KUKA KRL program: EPS_2_251674_SAN03_A_20251204014858.src

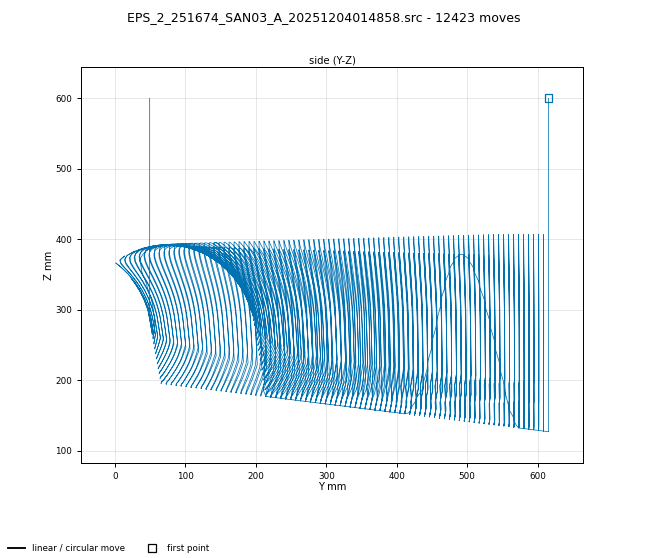
[picture p0: tool path of EPS_2_251674_SAN03_A_20251204014858.src, 12423 of 12425 moves have a stored position in this frame; points joined in program order, loops and branches not executed]
&ACCESS RVP
&REL 4
&COMMENT QRS 19112012
&PARAM EDITMASK = *
DEF PART()
EXT BAS (BAS_COMMAND :IN,REAL :IN )
INT I
BAS (#INITMOV,0 )

;KUKA QRS Post kuka4.cps  Date:22-06-2017 !

File_ID=2940

QRS_PRE_INIT()

;Init var - Until changes are made in qrs_pre_init
Outlet_Square_prg=0
Inlet_1_Square_prg=0
Inlet_2_Square_prg=0
Inlet_3_Square_prg=0
Inlet_4_Square_prg=0
Inlet_5_Square_prg=0

Outlet_1={X 0.000, Y 546.330, Z 306.500, B 0.000, E1 0.000 }
Inlet_1={X 0.000, Y 548.460, Z 276.500, B 0.000, E1 134.000 }
Outlet_1_type=201
Inlet_1_type=201
;QRS#1=Sidecore dimensions
;QRS#2=200-8" PVC SDR 35
;QRS#3=200-8" PVC SDR 35
;QRS#4=
;QRS#5=
;QRS#6=
;QRS#7=
;QRS#8=
;QRS#9=12-08 PSX
;QRS#10=12-08 PSX
;QRS#11=
;QRS#12=
;QRS#13=
;QRS#14=
;QRS#15=
;QRS#16=1220x127x686 2,25'
;QRS#17=EPS Height
;QRS#18=407
;QRS#19=*
;QRS#20= UPDATED VERSION 22-06-2017
;QRS#21=*
Outlet_Square=0100
Inlet_1_Square=0100
Inlet_2_Square=0
Inlet_3_Square=0
Inlet_4_Square=0
Inlet_5_Square=0
Mill_Square=1
Outlet_Square_Prg=204
Inlet_1_Square_prg=204

QRS_INIT()

$ADVANCE=5

; T1
PTP {E1 173.652,E2 173.652}
PTP {X 0,Y 615.437,A -85,B 0,C 180,E1 173.652,E2 173.652,E3 0,E4 0,E5 0,E6 0}
QRS_SPEED_INIT()
LIN {X 0,Y 615.437,Z 600,A -85,B 0,C 180,E1 173.652,E2 173.652,E3 0,E4 0,E5 0,E6 0} C_VEL
LIN {X 0,Y 615.437,Z 136.877,A -85,B 0,C 180,E1 173.652,E2 173.652} C_VEL
LIN {X 0,Y 615.437,Z 128.699,A -85,B 0,C 180,E1 173.652,E2 173.652} C_VEL
LIN {X 0,Y 615.423,Z 126.699,A -85,B 0,C 180,E1 173.466,E2 173.466} C_VEL
LIN {X 0,Y 615.421,Z 126.699,A -85,B 0,C 180,E1 171.463,E2 171.463} C_VEL
LIN {X 0,Y 615.417,Z 126.699,A -85,B 0,C 180,E1 169.141,E2 169.141} C_VEL
LIN {X 0,Y 615.44,Z 126.7,A -85,B 0,C 180,E1 166.798,E2 166.798} C_VEL
LIN {X 0,Y 615.461,Z 126.698,A -85,B 0,C 180,E1 164.094,E2 164.094} C_VEL
LIN {X 0,Y 615.415,Z 126.699,A -85,B 0,C 180,E1 161.352,E2 161.352} C_VEL
LIN {X 0,Y 615.494,Z 126.7,A -85,B 0,C 180,E1 158.569,E2 158.569} C_VEL
LIN {X 0,Y 615.418,Z 126.699,A -85,B 0,C 180,E1 155.725,E2 155.725} C_VEL
LIN {X 0,Y 615.429,Z 126.888,A -85,B 0,C 180,E1 155.186,E2 155.186} C_VEL
LIN {X 0,Y 615.495,Z 142.358,A -85,B 0,C 180,E1 152.64,E2 152.64} C_VEL
LIN {X 0,Y 615.484,Z 160.778,A -85,B 0,C 180,E1 149.651,E2 149.651} C_VEL
LIN {X 0,Y 615.49,Z 165.938,A -85,B 0,C 180,E1 148.82,E2 148.82} C_VEL
LIN {X 0,Y 615.49,Z 272.899,A -85,B 0,C 180,E1 147.543,E2 147.543} C_VEL
LIN {X 0,Y 615.48,Z 286.149,A -85,B 0,C 180,E1 147.251,E2 147.251} C_VEL
LIN {X 0,Y 615.485,Z 298.089,A -85,B 0,C 180,E1 146.862,E2 146.862} C_VEL
LIN {X 0,Y 615.469,Z 309.932,A -85,B 0,C 180,E1 146.343,E2 146.343} C_VEL
LIN {X 0,Y 615.468,Z 320.918,A -85,B 0,C 180,E1 145.722,E2 145.722} C_VEL
LIN {X 0,Y 615.498,Z 331.305,A -85,B 0,C 180,E1 144.987,E2 144.987} C_VEL
LIN {X 0,Y 615.497,Z 340.782,A -85,B 0,C 180,E1 144.164,E2 144.164} C_VEL
LIN {X 0,Y 615.498,Z 348.744,A -85,B 0,C 180,E1 143.319,E2 143.319} C_VEL
LIN {X 0,Y 615.496,Z 356.025,A -85,B 0,C 180,E1 142.373,E2 142.373} C_VEL
LIN {X 0,Y 615.493,Z 362.602,A -85,B 0,C 180,E1 141.306,E2 141.306} C_VEL
LIN {X 0,Y 615.493,Z 367.683,A -85,B 0,C 180,E1 140.251,E2 140.251} C_VEL
LIN {X 0,Y 615.494,Z 370.866,A -85,B 0,C 180,E1 139.394,E2 139.394} C_VEL
LIN {X 0,Y 615.496,Z 373.343,A -85,B 0,C 180,E1 138.527,E2 138.527} C_VEL
LIN {X 0,Y 615.499,Z 375.057,A -85,B 0,C 180,E1 137.648,E2 137.648} C_VEL
LIN {X 0,Y 615.498,Z 376.069,A -85,B 0,C 180,E1 136.757,E2 136.757} C_VEL
LIN {X 0,Y 615.496,Z 376.37,A -85,B 0,C 180,E1 135.852,E2 135.852} C_VEL
LIN {X 0,Y 615.496,Z 375.91,A -85,B 0,C 180,E1 134.933,E2 134.933} C_VEL
LIN {X 0,Y 615.493,Z 374.62,A -85,B 0,C 180,E1 133.998,E2 133.998} C_VEL
LIN {X 0,Y 615.494,Z 372.461,A -85,B 0,C 180,E1 133.048,E2 133.048} C_VEL
LIN {X 0,Y 615.497,Z 369.346,A -85,B 0,C 180,E1 132.082,E2 132.082} C_VEL
LIN {X 0,Y 615.494,Z 363.935,A -85,B 0,C 180,E1 130.85,E2 130.85} C_VEL
LIN {X 0,Y 615.498,Z 357.456,A -85,B 0,C 180,E1 129.748,E2 129.748} C_VEL
LIN {X 0,Y 615.496,Z 349.585,A -85,B 0,C 180,E1 128.693,E2 128.693} C_VEL
LIN {X 0,Y 615.498,Z 340.528,A -85,B 0,C 180,E1 127.723,E2 127.723} C_VEL
LIN {X 0,Y 615.495,Z 329.848,A -85,B 0,C 180,E1 126.809,E2 126.809} C_VEL
LIN {X 0,Y 615.465,Z 319.974,A -85,B 0,C 180,E1 126.127,E2 126.127} C_VEL
LIN {X 0,Y 615.469,Z 308.871,A -85,B 0,C 180,E1 125.516,E2 125.516} C_VEL
LIN {X 0,Y 615.483,Z 295.83,A -85,B 0,C 180,E1 124.964,E2 124.964} C_VEL
LIN {X 0,Y 615.48,Z 282.891,A -85,B 0,C 180,E1 124.572,E2 124.572} C_VEL
LIN {X 0,Y 615.483,Z 269.51,A -85,B 0,C 180,E1 124.317,E2 124.317} C_VEL
LIN {X 0,Y 615.483,Z 165.935,A -85,B 0,C 180,E1 123.089,E2 123.089} C_VEL
LIN {X 0,Y 615.492,Z 147.811,A -85,B 0,C 180,E1 120.159,E2 120.159} C_VEL
LIN {X 0,Y 615.493,Z 130.723,A -85,B 0,C 180,E1 117.36,E2 117.36} C_VEL
LIN {X 0,Y 615.428,Z 126.699,A -85,B 0,C 180,E1 116.67,E2 116.67} C_VEL
LIN {X 0,Y 615.421,Z 126.698,A -85,B 0,C 180,E1 114.274,E2 114.274} C_VEL
LIN {X 0,Y 615.498,Z 126.7,A -85,B 0,C 180,E1 111.431,E2 111.431} C_VEL
LIN {X 0,Y 615.419,Z 126.698,A -85,B 0,C 180,E1 108.587,E2 108.587} C_VEL
LIN {X 0,Y 615.463,Z 126.697,A -85,B 0,C 180,E1 105.905,E2 105.905} C_VEL
LIN {X 0,Y 615.446,Z 126.699,A -85,B 0,C 180,E1 103.202,E2 103.202} C_VEL
LIN {X 0,Y 615.421,Z 126.698,A -85,B 0,C 180,E1 100.858,E2 100.858} C_VEL
LIN {X 0,Y 615.424,Z 126.698,A -85,B 0,C 180,E1 98.537,E2 98.537} C_VEL
LIN {X 0,Y 615.496,Z 126.696,A -85,B 0,C 180,E1 95.898,E2 95.898} C_VEL
LIN {X 0,Y 615.433,Z 126.699,A -85,B 0,C 180,E1 93.273,E2 93.273} C_VEL
LIN {X 0,Y 615.432,Z 126.699,A -85,B 0,C 180,E1 91.309,E2 91.309} C_VEL
LIN {X 0,Y 615.431,Z 126.699,A -85,B 0,C 180,E1 89.346,E2 89.346} C_VEL
LIN {X 0,Y 615.431,Z 126.699,A -85,B 0,C 180,E1 87.382,E2 87.382} C_VEL
LIN {X 0,Y 615.429,Z 126.699,A -85,B 0,C 180,E1 85.415,E2 85.415} C_VEL
LIN {X 0,Y 615.429,Z 126.699,A -85,B 0,C 180,E1 83.443,E2 83.443} C_VEL
LIN {X 0,Y 615.428,Z 126.699,A -85,B 0,C 180,E1 81.463,E2 81.463} C_VEL
LIN {X 0,Y 615.417,Z 126.699,A -85,B 0,C 180,E1 79.145,E2 79.145} C_VEL
LIN {X 0,Y 615.437,Z 126.698,A -85,B 0,C 180,E1 76.798,E2 76.798} C_VEL
LIN {X 0,Y 615.47,Z 126.701,A -85,B 0,C 180,E1 74.094,E2 74.094} C_VEL
LIN {X 0,Y 615.419,Z 126.698,A -85,B 0,C 180,E1 71.352,E2 71.352} C_VEL
LIN {X 0,Y 615.486,Z 126.697,A -85,B 0,C 180,E1 68.568,E2 68.568} C_VEL
LIN {X 0,Y 615.423,Z 126.699,A -85,B 0,C 180,E1 65.726,E2 65.726} C_VEL
LIN {X 0,Y 615.417,Z 126.699,A -85,B 0,C 180,E1 63.553,E2 63.553} C_VEL
LIN {X 0,Y 615.489,Z 126.702,A -85,B 0,C 180,E1 60.594,E2 60.594} C_VEL
LIN {X 0,Y 615.456,Z 126.7,A -85,B 0,C 180,E1 58.313,E2 58.313} C_VEL
LIN {X 0,Y 615.424,Z 126.699,A -85,B 0,C 180,E1 55.974,E2 55.974} C_VEL
LIN {X 0,Y 615.422,Z 126.698,A -85,B 0,C 180,E1 53.571,E2 53.571} C_VEL
LIN {X 0,Y 615.489,Z 126.697,A -85,B 0,C 180,E1 50.937,E2 50.937} C_VEL
LIN {X 0,Y 615.455,Z 126.7,A -85,B 0,C 180,E1 48.524,E2 48.524} C_VEL
LIN {X 0,Y 615.418,Z 126.699,A -85,B 0,C 180,E1 46.009,E2 46.009} C_VEL
LIN {X 0,Y 615.418,Z 126.699,A -85,B 0,C 180,E1 43.991,E2 43.991} C_VEL
LIN {X 0,Y 615.446,Z 126.698,A -85,B 0,C 180,E1 41.477,E2 41.477} C_VEL
LIN {X 0,Y 615.476,Z 126.7,A -85,B 0,C 180,E1 38.905,E2 38.905} C_VEL
LIN {X 0,Y 615.424,Z 126.699,A -85,B 0,C 180,E1 36.429,E2 36.429} C_VEL
LIN {X 0,Y 615.42,Z 126.698,A -85,B 0,C 180,E1 34.026,E2 34.026} C_VEL
LIN {X 0,Y 615.444,Z 126.698,A -85,B 0,C 180,E1 31.688,E2 31.688} C_VEL
LIN {X 0,Y 615.478,Z 126.7,A -85,B 0,C 180,E1 29.406,E2 29.406} C_VEL
LIN {X 0,Y 615.418,Z 126.699,A -85,B 0,C 180,E1 26.447,E2 26.447} C_VEL
LIN {X 0,Y 615.433,Z 126.698,A -85,B 0,C 180,E1 23.999,E2 23.999} C_VEL
LIN {X 0,Y 615.497,Z 126.7,A -85,B 0,C 180,E1 21.431,E2 21.431} C_VEL
LIN {X 0,Y 615.415,Z 126.699,A -85,B 0,C 180,E1 18.587,E2 18.587} C_VEL
LIN {X 0,Y 615.462,Z 126.698,A -85,B 0,C 180,E1 15.906,E2 15.906} C_VEL
LIN {X 0,Y 615.442,Z 126.699,A -85,B 0,C 180,E1 13.202,E2 13.202} C_VEL
LIN {X 0,Y 615.417,Z 126.699,A -85,B 0,C 180,E1 10.858,E2 10.858} C_VEL
LIN {X 0,Y 615.422,Z 126.698,A -85,B 0,C 180,E1 8.537,E2 8.537} C_VEL
LIN {X 0,Y 615.496,Z 126.698,A -85,B 0,C 180,E1 5.898,E2 5.898} C_VEL
LIN {X 0,Y 615.429,Z 126.699,A -85,B 0,C 180,E1 3.273,E2 3.273} C_VEL
LIN {X 0,Y 615.429,Z 126.699,A -85,B 0,C 180,E1 1.308,E2 1.308} C_VEL
LIN {X 0,Y 615.428,Z 126.699,A -85,B 0,C 180,E1 -0.655,E2 -0.655} C_VEL
LIN {X 0,Y 615.428,Z 126.699,A -85,B 0,C 180,E1 -2.618,E2 -2.618} C_VEL
LIN {X 0,Y 615.426,Z 126.699,A -85,B 0,C 180,E1 -4.585,E2 -4.585} C_VEL
LIN {X 0,Y 615.426,Z 126.699,A -85,B 0,C 180,E1 -6.558,E2 -6.558} C_VEL
LIN {X 0,Y 615.425,Z 126.699,A -85,B 0,C 180,E1 -8.538,E2 -8.538} C_VEL
LIN {X 0,Y 615.423,Z 126.699,A -85,B 0,C 180,E1 -10.528,E2 -10.528} C_VEL
LIN {X 0,Y 615.421,Z 126.699,A -85,B 0,C 180,E1 -12.532,E2 -12.532} C_VEL
LIN {X 0,Y 615.418,Z 126.699,A -85,B 0,C 180,E1 -14.551,E2 -14.551} C_VEL
LIN {X 0,Y 615.416,Z 126.699,A -85,B 0,C 180,E1 -16.589,E2 -16.589} C_VEL
LIN {X 0,Y 615.465,Z 126.698,A -85,B 0,C 180,E1 -19.339,E2 -19.339} C_VEL
LIN {X 0,Y 615.43,Z 126.699,A -85,B 0,C 180,E1 -22.139,E2 -22.139} C_VEL
LIN {X 0,Y 615.42,Z 126.699,A -85,B 0,C 180,E1 -24.275,E2 -24.275} C_VEL
LIN {X 0,Y 615.414,Z 126.699,A -85,B 0,C 180,E1 -26.448,E2 -26.448} C_VEL
LIN {X 0,Y 615.485,Z 126.703,A -85,B 0,C 180,E1 -29.407,E2 -29.407} C_VEL
LIN {X 0,Y 615.452,Z 126.7,A -85,B 0,C 180,E1 -31.688,E2 -31.688} C_VEL
LIN {X 0,Y 615.421,Z 126.699,A -85,B 0,C 180,E1 -34.026,E2 -34.026} C_VEL
LIN {X 0,Y 615.42,Z 126.699,A -85,B 0,C 180,E1 -36.43,E2 -36.43} C_VEL
LIN {X 0,Y 615.489,Z 126.698,A -85,B 0,C 180,E1 -39.063,E2 -39.063} C_VEL
LIN {X 0,Y 615.451,Z 126.7,A -85,B 0,C 180,E1 -41.477,E2 -41.477} C_VEL
LIN {X 0,Y 615.416,Z 126.699,A -85,B 0,C 180,E1 -43.991,E2 -43.991} C_VEL
LIN {X 0,Y 615.414,Z 126.699,A -85,B 0,C 180,E1 -46.01,E2 -46.01} C_VEL
LIN {X 0,Y 615.445,Z 126.699,A -85,B 0,C 180,E1 -48.523,E2 -48.523} C_VEL
LIN {X 0,Y 615.472,Z 126.7,A -85,B 0,C 180,E1 -51.095,E2 -51.095} C_VEL
LIN {X 0,Y 615.421,Z 126.699,A -85,B 0,C 180,E1 -53.571,E2 -53.571} C_VEL
LIN {X 0,Y 615.418,Z 126.699,A -85,B 0,C 180,E1 -55.974,E2 -55.974} C_VEL
LIN {X 0,Y 615.443,Z 126.699,A -85,B 0,C 180,E1 -58.312,E2 -58.312} C_VEL
LIN {X 0,Y 615.477,Z 126.701,A -85,B 0,C 180,E1 -60.594,E2 -60.594} C_VEL
LIN {X 0,Y 615.415,Z 126.699,A -85,B 0,C 180,E1 -63.553,E2 -63.553} C_VEL
LIN {X 0,Y 615.433,Z 126.699,A -85,B 0,C 180,E1 -66.004,E2 -66.004} C_VEL
LIN {X 0,Y 615.424,Z 126.778,A -85,B 0,C 180,E1 -67.838,E2 -67.838} C_VEL
LIN {X 0,Y 615.497,Z 145.82,A -85,B 0,C 180,E1 -70.489,E2 -70.489} C_VEL
LIN {X 0,Y 615.458,Z 165.932,A -85,B 0,C 180,E1 -73.242,E2 -73.242} C_VEL
LIN {X 0,Y 615.475,Z 185.71,A -85,B 0,C 180,E1 -75.916,E2 -75.916} C_VEL
LIN {X 0,Y 615.46,Z 194.645,A -85,B 0,C 180,E1 -77.113,E2 -77.113} C_VEL
LIN {X 0,Y 615.488,Z 302.833,A -85,B 0,C 180,E1 -78.411,E2 -78.411} C_VEL
LIN {X 0,Y 615.477,Z 315.348,A -85,B 0,C 180,E1 -78.682,E2 -78.682} C_VEL
LIN {X 0,Y 615.488,Z 328.618,A -85,B 0,C 180,E1 -79.113,E2 -79.113} C_VEL
LIN {X 0,Y 615.477,Z 340.48,A -85,B 0,C 180,E1 -79.639,E2 -79.639} C_VEL
LIN {X 0,Y 615.494,Z 351.994,A -85,B 0,C 180,E1 -80.304,E2 -80.304} C_VEL
LIN {X 0,Y 615.499,Z 362.341,A -85,B 0,C 180,E1 -81.05,E2 -81.05} C_VEL
LIN {X 0,Y 615.497,Z 370.812,A -85,B 0,C 180,E1 -81.794,E2 -81.794} C_VEL
LIN {X 0,Y 615.498,Z 378.606,A -85,B 0,C 180,E1 -82.62,E2 -82.62} C_VEL
LIN {X 0,Y 615.496,Z 386.203,A -85,B 0,C 180,E1 -83.608,E2 -83.608} C_VEL
LIN {X 0,Y 615.498,Z 393.204,A -85,B 0,C 180,E1 -84.759,E2 -84.759} C_VEL
LIN {X 0,Y 615.494,Z 397.851,A -85,B 0,C 180,E1 -85.744,E2 -85.744} C_VEL
LIN {X 0,Y 615.494,Z 401.398,A -85,B 0,C 180,E1 -86.727,E2 -86.727} C_VEL
LIN {X 0,Y 615.497,Z 403.233,A -85,B 0,C 180,E1 -87.382,E2 -87.382} C_VEL
LIN {X 0,Y 615.5,Z 404.607,A -85,B 0,C 180,E1 -88.037,E2 -88.037} C_VEL
LIN {X 0,Y 615.496,Z 406.173,A -85,B 0,C 180,E1 -89.346,E2 -89.346} C_VEL
LIN {X 0,Y 615.494,Z 406.389,A -85,B 0,C 180,E1 -90,E2 -90} C_VEL
LIN {X 0,Y 615.495,Z 405.58,A -85,B 0,C 180,E1 -91.308,E2 -91.308} C_VEL
LIN {X 0,Y 615.5,Z 404.608,A -85,B 0,C 180,E1 -91.963,E2 -91.963} C_VEL
LIN {X 0,Y 615.497,Z 403.233,A -85,B 0,C 180,E1 -92.618,E2 -92.618} C_VEL
LIN {X 0,Y 615.496,Z 400.35,A -85,B 0,C 180,E1 -93.6,E2 -93.6} C_VEL
LIN {X 0,Y 615.498,Z 396.442,A -85,B 0,C 180,E1 -94.584,E2 -94.584} C_VEL
LIN {X 0,Y 615.499,Z 391.406,A -85,B 0,C 180,E1 -95.569,E2 -95.569} C_VEL
LIN {X 0,Y 615.497,Z 384.87,A -85,B 0,C 180,E1 -96.583,E2 -96.583} C_VEL
LIN {X 0,Y 615.497,Z 377.135,A -85,B 0,C 180,E1 -97.545,E2 -97.545} C_VEL
LIN {X 0,Y 615.498,Z 369.047,A -85,B 0,C 180,E1 -98.371,E2 -98.371} C_VEL
LIN {X 0,Y 615.499,Z 359.171,A -85,B 0,C 180,E1 -99.198,E2 -99.198} C_VEL
LIN {X 0,Y 615.488,Z 347.986,A -85,B 0,C 180,E1 -99.945,E2 -99.945} C_VEL
LIN {X 0,Y 615.482,Z 337.029,A -85,B 0,C 180,E1 -100.527,E2 -100.527} C_VEL
LIN {X 0,Y 615.48,Z 324.495,A -85,B 0,C 180,E1 -101.04,E2 -101.04} C_VEL
LIN {X 0,Y 615.479,Z 312.079,A -85,B 0,C 180,E1 -101.401,E2 -101.401} C_VEL
LIN {X 0,Y 615.493,Z 298.485,A -85,B 0,C 180,E1 -101.652,E2 -101.652} C_VEL
LIN {X 0,Y 615.46,Z 194.647,A -85,B 0,C 180,E1 -102.887,E2 -102.887} C_VEL
LIN {X 0,Y 615.497,Z 173.467,A -85,B 0,C 180,E1 -105.735,E2 -105.735} C_VEL
LIN {X 0,Y 615.482,Z 152.11,A -85,B 0,C 180,E1 -108.646,E2 -108.646} C_VEL
LIN {X 0,Y 615.494,Z 131.984,A -85,B 0,C 180,E1 -111.431,E2 -111.431} C_VEL
LIN {X 0,Y 615.423,Z 126.699,A -85,B 0,C 180,E1 -112.186,E2 -112.186} C_VEL
LIN {X 0,Y 615.417,Z 126.699,A -85,B 0,C 180,E1 -114.274,E2 -114.274} C_VEL
LIN {X 0,Y 615.415,Z 126.699,A -85,B 0,C 180,E1 -116.447,E2 -116.447} C_VEL
LIN {X 0,Y 615.478,Z 126.701,A -85,B 0,C 180,E1 -119.406,E2 -119.406} C_VEL
LIN {X 0,Y 615.446,Z 126.699,A -85,B 0,C 180,E1 -121.687,E2 -121.687} C_VEL
LIN {X 0,Y 615.418,Z 126.699,A -85,B 0,C 180,E1 -124.026,E2 -124.026} C_VEL
LIN {X 0,Y 615.465,Z 126.701,A -85,B 0,C 180,E1 -126.933,E2 -126.933} C_VEL
LIN {X 0,Y 615.423,Z 126.699,A -85,B 0,C 180,E1 -129.754,E2 -129.754} C_VEL
LIN {X 0,Y 615.415,Z 126.699,A -85,B 0,C 180,E1 -132.072,E2 -132.072} C_VEL
LIN {X 0,Y 615.416,Z 126.7,A -85,B 0,C 180,E1 -134.155,E2 -134.155} C_VEL
LIN {X 0,Y 615.475,Z 126.7,A -85,B 0,C 180,E1 -136.754,E2 -136.754} C_VEL
LIN {X 0,Y 615.437,Z 126.699,A -85,B 0,C 180,E1 -139.389,E2 -139.389} C_VEL
LIN {X 0,Y 615.465,Z 126.698,A -85,B 0,C 180,E1 -141.094,E2 -141.094} C_VEL
LIN {X 0,Y 615.419,Z 126.699,A -85,B 0,C 180,E1 -143.57,E2 -143.57} C_VEL
LIN {X 0,Y 615.465,Z 126.7,A -85,B 0,C 180,E1 -146.468,E2 -146.468} C_VEL
LIN {X 0,Y 615.446,Z 126.699,A -85,B 0,C 180,E1 -149.078,E2 -149.078} C_VEL
LIN {X 0,Y 615.415,Z 126.699,A -85,B 0,C 180,E1 -151.56,E2 -151.56} C_VEL
LIN {X 0,Y 615.463,Z 126.7,A -85,B 0,C 180,E1 -154.283,E2 -154.283} C_VEL
LIN {X 0,Y 615.425,Z 126.699,A -85,B 0,C 180,E1 -157.153,E2 -157.153} C_VEL
LIN {X 0,Y 615.415,Z 126.699,A -85,B 0,C 180,E1 -159.458,E2 -159.458} C_VEL
LIN {X 0,Y 615.451,Z 126.701,A -85,B 0,C 180,E1 -162.042,E2 -162.042} C_VEL
LIN {X 0,Y 615.442,Z 126.699,A -85,B 0,C 180,E1 -164.773,E2 -164.773} C_VEL
LIN {X 0,Y 615.435,Z 126.699,A -85,B 0,C 180,E1 -166.797,E2 -166.797} C_VEL
LIN {X 0,Y 615.416,Z 126.699,A -85,B 0,C 180,E1 -169.142,E2 -169.142} C_VEL
LIN {X 0,Y 615.423,Z 126.699,A -85,B 0,C 180,E1 -171.462,E2 -171.462} C_VEL
LIN {X 0,Y 615.498,Z 126.7,A -85,B 0,C 180,E1 -174.101,E2 -174.101} C_VEL
LIN {X 0,Y 615.425,Z 126.699,A -85,B 0,C 180,E1 -176.726,E2 -176.726} C_VEL
LIN {X 0,Y 615.423,Z 126.699,A -85,B 0,C 180,E1 -178.691,E2 -178.691} C_VEL
LIN {X 0,Y 615.424,Z 126.699,A -85,B 0,C 180,E1 -180.654,E2 -180.654} C_VEL
LIN {X 0,Y 615.423,Z 126.699,A -85,B 0,C 180,E1 -182.618,E2 -182.618} C_VEL
LIN {X 0,Y 615.423,Z 126.699,A -85,B 0,C 180,E1 -184.585,E2 -184.585} C_VEL
LIN {X 0,Y 615.423,Z 126.699,A -85,B 0,C 180,E1 -186.534,E2 -186.534} C_VEL
LIN {X 0,Y 614.749,Z 126.846,A -85,B 0,C 180,E1 -187.08,E2 -187.08} C_VEL
LIN {X 0,Y 611.916,Z 127.263,A -85,B 0,C 180,E1 -187.967,E2 -187.967} C_VEL
LIN {X 0,Y 609.531,Z 127.57,A -85,B 0,C 180,E1 -188.679,E2 -188.679} C_VEL
LIN {X 0,Y 608.508,Z 127.685,A -85,B 0,C 180,E1 -189.229,E2 -189.229} C_VEL
LIN {X 0,Y 608.425,Z 127.694,A -85,B 0,C 180,E1 -189.415,E2 -189.415} C_VEL
LIN {X 0,Y 608.44,Z 127.694,A -85,B 0,C 180,E1 -192,E2 -192} C_VEL
LIN {X 0,Y 608.388,Z 127.696,A -85,B 0,C 180,E1 -194.722,E2 -194.722} C_VEL
LIN {X 0,Y 608.421,Z 127.701,A -85,B 0,C 180,E1 -197.477,E2 -197.477} C_VEL
LIN {X 0,Y 608.406,Z 127.694,A -85,B 0,C 180,E1 -200.276,E2 -200.276} C_VEL
LIN {X 0,Y 608.387,Z 127.696,A -85,B 0,C 180,E1 -202.462,E2 -202.462} C_VEL
LIN {X 0,Y 608.432,Z 127.813,A -85,B 0,C 180,E1 -204.731,E2 -204.731} C_VEL
LIN {X 0,Y 608.495,Z 142.748,A -85,B 0,C 180,E1 -207.212,E2 -207.212} C_VEL
LIN {X 0,Y 608.461,Z 159.611,A -85,B 0,C 180,E1 -209.972,E2 -209.972} C_VEL
LIN {X 0,Y 608.46,Z 166.158,A -85,B 0,C 180,E1 -211.035,E2 -211.035} C_VEL
LIN {X 0,Y 608.536,Z 273.771,A -85,B 0,C 180,E1 -212.336,E2 -212.336} C_VEL
LIN {X 0,Y 608.53,Z 287.37,A -85,B 0,C 180,E1 -212.649,E2 -212.649} C_VEL
LIN {X 0,Y 608.528,Z 299.804,A -85,B 0,C 180,E1 -213.072,E2 -213.072} C_VEL
LIN {X 0,Y 608.482,Z 310.749,A -85,B 0,C 180,E1 -213.57,E2 -213.57} C_VEL
LIN {X 0,Y 608.479,Z 321.147,A -85,B 0,C 180,E1 -214.167,E2 -214.167} C_VEL
LIN {X 0,Y 608.489,Z 331.59,A -85,B 0,C 180,E1 -214.912,E2 -214.912} C_VEL
LIN {X 0,Y 608.459,Z 340.46,A -85,B 0,C 180,E1 -215.683,E2 -215.683} C_VEL
LIN {X 0,Y 608.454,Z 348.278,A -85,B 0,C 180,E1 -216.502,E2 -216.502} C_VEL
LIN {X 0,Y 608.443,Z 356.667,A -85,B 0,C 180,E1 -217.586,E2 -217.586} C_VEL
LIN {X 0,Y 608.454,Z 362.837,A -85,B 0,C 180,E1 -218.589,E2 -218.589} C_VEL
LIN {X 0,Y 608.425,Z 367.101,A -85,B 0,C 180,E1 -219.443,E2 -219.443} C_VEL
LIN {X 0,Y 608.425,Z 370.632,A -85,B 0,C 180,E1 -220.327,E2 -220.327} C_VEL
LIN {X 0,Y 608.422,Z 373.658,A -85,B 0,C 180,E1 -221.339,E2 -221.339} C_VEL
LIN {X 0,Y 608.439,Z 375.657,A -85,B 0,C 180,E1 -222.333,E2 -222.333} C_VEL
LIN {X 0,Y 608.434,Z 376.73,A -85,B 0,C 180,E1 -223.306,E2 -223.306} C_VEL
LIN {X 0,Y 608.419,Z 376.955,A -85,B 0,C 180,E1 -224.261,E2 -224.261} C_VEL
LIN {X 0,Y 608.418,Z 376.38,A -85,B 0,C 180,E1 -225.202,E2 -225.202} C_VEL
LIN {X 0,Y 608.426,Z 375.036,A -85,B 0,C 180,E1 -226.128,E2 -226.128} C_VEL
LIN {X 0,Y 608.435,Z 372.887,A -85,B 0,C 180,E1 -227.04,E2 -227.04} C_VEL
LIN {X 0,Y 608.429,Z 369.983,A -85,B 0,C 180,E1 -227.937,E2 -227.937} C_VEL
LIN {X 0,Y 608.439,Z 365.231,A -85,B 0,C 180,E1 -229.043,E2 -229.043} C_VEL
LIN {X 0,Y 608.44,Z 359.156,A -85,B 0,C 180,E1 -230.129,E2 -230.129} C_VEL
LIN {X 0,Y 608.468,Z 352.63,A -85,B 0,C 180,E1 -231.06,E2 -231.06} C_VEL
LIN {X 0,Y 608.454,Z 344.456,A -85,B 0,C 180,E1 -232.008,E2 -232.008} C_VEL
LIN {X 0,Y 608.467,Z 334.283,A -85,B 0,C 180,E1 -232.962,E2 -232.962} C_VEL
LIN {X 0,Y 608.487,Z 324.432,A -85,B 0,C 180,E1 -233.706,E2 -233.706} C_VEL
LIN {X 0,Y 608.483,Z 314.487,A -85,B 0,C 180,E1 -234.319,E2 -234.319} C_VEL
LIN {X 0,Y 608.517,Z 302.84,A -85,B 0,C 180,E1 -234.89,E2 -234.89} C_VEL
LIN {X 0,Y 608.508,Z 290.071,A -85,B 0,C 180,E1 -235.362,E2 -235.362} C_VEL
LIN {X 0,Y 608.535,Z 276.745,A -85,B 0,C 180,E1 -235.699,E2 -235.699} C_VEL
LIN {X 0,Y 608.548,Z 258.935,A -85,B 0,C 180,E1 -235.949,E2 -235.949} C_VEL
LIN {X 0,Y 608.466,Z 166.127,A -85,B 0,C 180,E1 -237.06,E2 -237.06} C_VEL
LIN {X 0,Y 608.477,Z 149.448,A -85,B 0,C 180,E1 -239.777,E2 -239.777} C_VEL
LIN {X 0,Y 608.504,Z 133.038,A -85,B 0,C 180,E1 -242.485,E2 -242.485} C_VEL
LIN {X 0,Y 608.405,Z 127.695,A -85,B 0,C 180,E1 -243.409,E2 -243.409} C_VEL
LIN {X 0,Y 608.432,Z 127.693,A -85,B 0,C 180,E1 -246.154,E2 -246.154} C_VEL
LIN {X 0,Y 608.428,Z 127.694,A -85,B 0,C 180,E1 -249.018,E2 -249.018} C_VEL
LIN {X 0,Y 608.403,Z 127.695,A -85,B 0,C 180,E1 -251.827,E2 -251.827} C_VEL
LIN {X 0,Y 608.443,Z 127.697,A -85,B 0,C 180,E1 -254.594,E2 -254.594} C_VEL
LIN {X 0,Y 608.395,Z 127.695,A -85,B 0,C 180,E1 -257.322,E2 -257.322} C_VEL
LIN {X 0,Y 608.446,Z 127.694,A -85,B 0,C 180,E1 -260.023,E2 -260.023} C_VEL
LIN {X 0,Y 608.415,Z 127.696,A -85,B 0,C 180,E1 -262.7,E2 -262.7} C_VEL
LIN {X 0,Y 608.422,Z 127.694,A -85,B 0,C 180,E1 -264.698,E2 -264.698} C_VEL
LIN {X 0,Y 608.422,Z 127.692,A -85,B 0,C 180,E1 -267.352,E2 -267.352} C_VEL
LIN {X 0,Y 608.472,Z 127.694,A -85,B 0,C 180,E1 -270,E2 -270} C_VEL
LIN {X 0,Y 608.426,Z 127.692,A -85,B 0,C 180,E1 -272.648,E2 -272.648} C_VEL
LIN {X 0,Y 608.414,Z 127.693,A -85,B 0,C 180,E1 -275.302,E2 -275.302} C_VEL
LIN {X 0,Y 608.466,Z 127.696,A -85,B 0,C 180,E1 -277.967,E2 -277.967} C_VEL
LIN {X 0,Y 608.402,Z 127.694,A -85,B 0,C 180,E1 -280.651,E2 -280.651} C_VEL
LIN {X 0,Y 608.428,Z 127.694,A -85,B 0,C 180,E1 -283.357,E2 -283.357} C_VEL
LIN {X 0,Y 608.428,Z 127.695,A -85,B 0,C 180,E1 -286.095,E2 -286.095} C_VEL
LIN {X 0,Y 608.423,Z 127.692,A -85,B 0,C 180,E1 -288.87,E2 -288.87} C_VEL
LIN {X 0,Y 608.449,Z 127.697,A -85,B 0,C 180,E1 -291.692,E2 -291.692} C_VEL
LIN {X 0,Y 608.406,Z 127.693,A -85,B 0,C 180,E1 -294.573,E2 -294.573} C_VEL
LIN {X 0,Y 608.458,Z 127.693,A -85,B 0,C 180,E1 -297.204,E2 -297.204} C_VEL
LIN {X 0,Y 608.409,Z 127.695,A -85,B 0,C 180,E1 -299.962,E2 -299.962} C_VEL
LIN {X 0,Y 608.406,Z 127.694,A -85,B 0,C 180,E1 -302.515,E2 -302.515} C_VEL
LIN {X 0,Y 608.412,Z 127.696,A -85,B 0,C 180,E1 -304.901,E2 -304.901} C_VEL
LIN {X 0,Y 608.43,Z 127.693,A -85,B 0,C 180,E1 -307.749,E2 -307.749} C_VEL
LIN {X 0,Y 608.395,Z 127.695,A -85,B 0,C 180,E1 -310.323,E2 -310.323} C_VEL
LIN {X 0,Y 608.44,Z 127.697,A -85,B 0,C 180,E1 -312.96,E2 -312.96} C_VEL
LIN {X 0,Y 608.403,Z 127.695,A -85,B 0,C 180,E1 -315.741,E2 -315.741} C_VEL
LIN {X 0,Y 608.402,Z 127.694,A -85,B 0,C 180,E1 -317.934,E2 -317.934} C_VEL
LIN {X 0,Y 608.432,Z 127.696,A -85,B 0,C 180,E1 -320.706,E2 -320.706} C_VEL
LIN {X 0,Y 608.442,Z 127.696,A -85,B 0,C 180,E1 -323.084,E2 -323.084} C_VEL
LIN {X 0,Y 608.422,Z 127.692,A -85,B 0,C 180,E1 -325.528,E2 -325.528} C_VEL
LIN {X 0,Y 608.412,Z 127.693,A -85,B 0,C 180,E1 -327.903,E2 -327.903} C_VEL
LIN {X 0,Y 608.427,Z 127.693,A -85,B 0,C 180,E1 -330.219,E2 -330.219} C_VEL
LIN {X 0,Y 608.464,Z 127.695,A -85,B 0,C 180,E1 -332.794,E2 -332.794} C_VEL
LIN {X 0,Y 608.404,Z 127.694,A -85,B 0,C 180,E1 -335.427,E2 -335.427} C_VEL
LIN {X 0,Y 608.453,Z 127.694,A -85,B 0,C 180,E1 -338.308,E2 -338.308} C_VEL
LIN {X 0,Y 608.403,Z 127.694,A -85,B 0,C 180,E1 -341.301,E2 -341.301} C_VEL
LIN {X 0,Y 608.422,Z 127.694,A -85,B 0,C 180,E1 -343.905,E2 -343.905} C_VEL
LIN {X 0,Y 608.429,Z 127.696,A -85,B 0,C 180,E1 -346.643,E2 -346.643} C_VEL
LIN {X 0,Y 608.4,Z 127.694,A -85,B 0,C 180,E1 -349.349,E2 -349.349} C_VEL
LIN {X 0,Y 608.463,Z 127.693,A -85,B 0,C 180,E1 -352.033,E2 -352.033} C_VEL
LIN {X 0,Y 608.418,Z 127.694,A -85,B 0,C 180,E1 -354.698,E2 -354.698} C_VEL
LIN {X 0,Y 608.42,Z 127.692,A -85,B 0,C 180,E1 -357.352,E2 -357.352} C_VEL
LIN {X 0,Y 608.469,Z 127.695,A -85,B 0,C 180,E1 -360,E2 -360} C_VEL
LIN {X 0,Y 608.423,Z 127.693,A -85,B 0,C 180,E1 -362.649,E2 -362.649} C_VEL
LIN {X 0,Y 608.413,Z 127.694,A -85,B 0,C 180,E1 -365.303,E2 -365.303} C_VEL
LIN {X 0,Y 608.463,Z 127.695,A -85,B 0,C 180,E1 -367.967,E2 -367.967} C_VEL
LIN {X 0,Y 608.402,Z 127.694,A -85,B 0,C 180,E1 -370.651,E2 -370.651} C_VEL
LIN {X 0,Y 608.426,Z 127.695,A -85,B 0,C 180,E1 -373.358,E2 -373.358} C_VEL
LIN {X 0,Y 608.427,Z 127.695,A -85,B 0,C 180,E1 -376.095,E2 -376.095} C_VEL
LIN {X 0,Y 608.421,Z 127.692,A -85,B 0,C 180,E1 -378.871,E2 -378.871} C_VEL
LIN {X 0,Y 608.448,Z 127.697,A -85,B 0,C 180,E1 -381.693,E2 -381.693} C_VEL
LIN {X 0,Y 608.404,Z 127.693,A -85,B 0,C 180,E1 -384.573,E2 -384.573} C_VEL
LIN {X 0,Y 608.457,Z 127.693,A -85,B 0,C 180,E1 -387.205,E2 -387.205} C_VEL
LIN {X 0,Y 608.405,Z 127.695,A -85,B 0,C 180,E1 -389.963,E2 -389.963} C_VEL
LIN {X 0,Y 608.404,Z 127.694,A -85,B 0,C 180,E1 -392.515,E2 -392.515} C_VEL
LIN {X 0,Y 608.411,Z 127.697,A -85,B 0,C 180,E1 -394.901,E2 -394.901} C_VEL
LIN {X 0,Y 608.428,Z 127.693,A -85,B 0,C 180,E1 -397.75,E2 -397.75} C_VEL
LIN {X 0,Y 608.398,Z 127.695,A -85,B 0,C 180,E1 -400.324,E2 -400.324} C_VEL
LIN {X 0,Y 608.438,Z 127.698,A -85,B 0,C 180,E1 -402.961,E2 -402.961} C_VEL
LIN {X 0,Y 608.399,Z 127.695,A -85,B 0,C 180,E1 -405.742,E2 -405.742} C_VEL
LIN {X 0,Y 608.4,Z 127.694,A -85,B 0,C 180,E1 -407.934,E2 -407.934} C_VEL
LIN {X 0,Y 608.433,Z 127.697,A -85,B 0,C 180,E1 -410.707,E2 -410.707} C_VEL
LIN {X 0,Y 608.437,Z 127.696,A -85,B 0,C 180,E1 -413.084,E2 -413.084} C_VEL
LIN {X 0,Y 608.42,Z 127.692,A -85,B 0,C 180,E1 -415.528,E2 -415.528} C_VEL
LIN {X 0,Y 608.41,Z 127.693,A -85,B 0,C 180,E1 -417.903,E2 -417.903} C_VEL
LIN {X 0,Y 608.426,Z 127.694,A -85,B 0,C 180,E1 -420.219,E2 -420.219} C_VEL
LIN {X 0,Y 608.463,Z 127.694,A -85,B 0,C 180,E1 -422.796,E2 -422.796} C_VEL
LIN {X 0,Y 608.405,Z 127.694,A -85,B 0,C 180,E1 -425.427,E2 -425.427} C_VEL
LIN {X 0,Y 608.426,Z 127.892,A -85,B 0,C 180,E1 -427.727,E2 -427.727} C_VEL
LIN {X 0,Y 608.533,Z 142.059,A -85,B 0,C 180,E1 -429.729,E2 -429.729} C_VEL
LIN {X 0,Y 608.515,Z 160.949,A -85,B 0,C 180,E1 -432.352,E2 -432.352} C_VEL
LIN {X 0,Y 608.488,Z 182.357,A -85,B 0,C 180,E1 -435.28,E2 -435.28} C_VEL
LIN {X 0,Y 608.467,Z 195.149,A -85,B 0,C 180,E1 -436.984,E2 -436.984} C_VEL
LIN {X 0,Y 608.547,Z 302.95,A -85,B 0,C 180,E1 -438.277,E2 -438.277} C_VEL
LIN {X 0,Y 608.512,Z 316.219,A -85,B 0,C 180,E1 -438.572,E2 -438.572} C_VEL
LIN {X 0,Y 608.513,Z 328.154,A -85,B 0,C 180,E1 -438.964,E2 -438.964} C_VEL
LIN {X 0,Y 608.499,Z 340.635,A -85,B 0,C 180,E1 -439.519,E2 -439.519} C_VEL
LIN {X 0,Y 608.484,Z 352.198,A -85,B 0,C 180,E1 -440.191,E2 -440.191} C_VEL
LIN {X 0,Y 608.485,Z 362.594,A -85,B 0,C 180,E1 -440.946,E2 -440.946} C_VEL
LIN {X 0,Y 608.475,Z 371.112,A -85,B 0,C 180,E1 -441.699,E2 -441.699} C_VEL
LIN {X 0,Y 608.471,Z 378.96,A -85,B 0,C 180,E1 -442.534,E2 -442.534} C_VEL
LIN {X 0,Y 608.461,Z 386.287,A -85,B 0,C 180,E1 -443.485,E2 -443.485} C_VEL
LIN {X 0,Y 608.451,Z 391.866,A -85,B 0,C 180,E1 -444.366,E2 -444.366} C_VEL
LIN {X 0,Y 608.432,Z 396.95,A -85,B 0,C 180,E1 -445.362,E2 -445.362} C_VEL
LIN {X 0,Y 608.449,Z 400.896,A -85,B 0,C 180,E1 -446.358,E2 -446.358} C_VEL
LIN {X 0,Y 608.425,Z 403.809,A -85,B 0,C 180,E1 -447.352,E2 -447.352} C_VEL
LIN {X 0,Y 608.445,Z 405.201,A -85,B 0,C 180,E1 -448.014,E2 -448.014} C_VEL
LIN {X 0,Y 608.438,Z 406.783,A -85,B 0,C 180,E1 -449.338,E2 -449.338} C_VEL
LIN {X 0,Y 608.434,Z 407,A -85,B 0,C 180,E1 -450,E2 -450} C_VEL
LIN {X 0,Y 608.448,Z 406.184,A -85,B 0,C 180,E1 -451.324,E2 -451.324} C_VEL
LIN {X 0,Y 608.445,Z 405.202,A -85,B 0,C 180,E1 -451.986,E2 -451.986} C_VEL
LIN {X 0,Y 608.425,Z 403.81,A -85,B 0,C 180,E1 -452.648,E2 -452.648} C_VEL
LIN {X 0,Y 608.449,Z 400.897,A -85,B 0,C 180,E1 -453.642,E2 -453.642} C_VEL
LIN {X 0,Y 608.432,Z 396.951,A -85,B 0,C 180,E1 -454.638,E2 -454.638} C_VEL
LIN {X 0,Y 608.438,Z 390.878,A -85,B 0,C 180,E1 -455.801,E2 -455.801} C_VEL
LIN {X 0,Y 608.462,Z 384.237,A -85,B 0,C 180,E1 -456.799,E2 -456.799} C_VEL
LIN {X 0,Y 608.456,Z 375.991,A -85,B 0,C 180,E1 -457.8,E2 -457.8} C_VEL
LIN {X 0,Y 608.472,Z 367.539,A -85,B 0,C 180,E1 -458.636,E2 -458.636} C_VEL
LIN {X 0,Y 608.479,Z 357.094,A -85,B 0,C 180,E1 -459.473,E2 -459.473} C_VEL
LIN {X 0,Y 608.489,Z 346.76,A -85,B 0,C 180,E1 -460.145,E2 -460.145} C_VEL
LIN {X 0,Y 608.519,Z 335.271,A -85,B 0,C 180,E1 -460.74,E2 -460.74} C_VEL
LIN {X 0,Y 608.528,Z 322.898,A -85,B 0,C 180,E1 -461.224,E2 -461.224} C_VEL
LIN {X 0,Y 608.544,Z 309.451,A -85,B 0,C 180,E1 -461.596,E2 -461.596} C_VEL
LIN {X 0,Y 608.553,Z 297.106,A -85,B 0,C 180,E1 -461.807,E2 -461.807} C_VEL
LIN {X 0,Y 608.468,Z 195.168,A -85,B 0,C 180,E1 -463.016,E2 -463.016} C_VEL
LIN {X 0,Y 608.477,Z 177.322,A -85,B 0,C 180,E1 -465.405,E2 -465.405} C_VEL
LIN {X 0,Y 608.492,Z 157.173,A -85,B 0,C 180,E1 -468.17,E2 -468.17} C_VEL
LIN {X 0,Y 608.524,Z 139.854,A -85,B 0,C 180,E1 -470.581,E2 -470.581} C_VEL
LIN {X 0,Y 608.411,Z 127.736,A -85,B 0,C 180,E1 -472.296,E2 -472.296} C_VEL
LIN {X 0,Y 608.405,Z 127.694,A -85,B 0,C 180,E1 -474.573,E2 -474.573} C_VEL
LIN {X 0,Y 608.46,Z 127.695,A -85,B 0,C 180,E1 -477.203,E2 -477.203} C_VEL
LIN {X 0,Y 608.402,Z 127.695,A -85,B 0,C 180,E1 -479.96,E2 -479.96} C_VEL
LIN {X 0,Y 608.405,Z 127.694,A -85,B 0,C 180,E1 -482.514,E2 -482.514} C_VEL
LIN {X 0,Y 608.414,Z 127.698,A -85,B 0,C 180,E1 -484.9,E2 -484.9} C_VEL
LIN {X 0,Y 608.425,Z 127.692,A -85,B 0,C 180,E1 -487.749,E2 -487.749} C_VEL
LIN {X 0,Y 608.398,Z 127.695,A -85,B 0,C 180,E1 -490.323,E2 -490.323} C_VEL
LIN {X 0,Y 608.44,Z 127.699,A -85,B 0,C 180,E1 -492.96,E2 -492.96} C_VEL
LIN {X 0,Y 608.399,Z 127.695,A -85,B 0,C 180,E1 -495.741,E2 -495.741} C_VEL
LIN {X 0,Y 608.4,Z 127.694,A -85,B 0,C 180,E1 -497.933,E2 -497.933} C_VEL
LIN {X 0,Y 608.431,Z 127.699,A -85,B 0,C 180,E1 -500.706,E2 -500.706} C_VEL
LIN {X 0,Y 608.432,Z 127.695,A -85,B 0,C 180,E1 -503.083,E2 -503.083} C_VEL
LIN {X 0,Y 608.418,Z 127.692,A -85,B 0,C 180,E1 -505.527,E2 -505.527} C_VEL
LIN {X 0,Y 608.412,Z 127.693,A -85,B 0,C 180,E1 -507.902,E2 -507.902} C_VEL
LIN {X 0,Y 608.43,Z 127.694,A -85,B 0,C 180,E1 -510.218,E2 -510.218} C_VEL
LIN {X 0,Y 608.395,Z 127.696,A -85,B 0,C 180,E1 -513.223,E2 -513.223} C_VEL
LIN {X 0,Y 608.403,Z 127.694,A -85,B 0,C 180,E1 -515.427,E2 -515.427} C_VEL
LIN {X 0,Y 608.447,Z 127.696,A -85,B 0,C 180,E1 -518.307,E2 -518.307} C_VEL
LIN {X 0,Y 608.403,Z 127.694,A -85,B 0,C 180,E1 -521.3,E2 -521.3} C_VEL
LIN {X 0,Y 608.426,Z 127.695,A -85,B 0,C 180,E1 -523.905,E2 -523.905} C_VEL
LIN {X 0,Y 608.425,Z 127.695,A -85,B 0,C 180,E1 -526.642,E2 -526.642} C_VEL
LIN {X 0,Y 608.401,Z 127.694,A -85,B 0,C 180,E1 -529.349,E2 -529.349} C_VEL
LIN {X 0,Y 608.462,Z 127.695,A -85,B 0,C 180,E1 -532.033,E2 -532.033} C_VEL
LIN {X 0,Y 608.412,Z 127.694,A -85,B 0,C 180,E1 -534.697,E2 -534.697} C_VEL
LIN {X 0,Y 608.421,Z 127.693,A -85,B 0,C 180,E1 -537.351,E2 -537.351} C_VEL
LIN {X 0,Y 608.468,Z 127.695,A -85,B 0,C 180,E1 -540,E2 -540} C_VEL
LIN {X 0,Y 608.419,Z 127.692,A -85,B 0,C 180,E1 -542.648,E2 -542.648} C_VEL
LIN {X 0,Y 608.417,Z 127.694,A -85,B 0,C 180,E1 -545.302,E2 -545.302} C_VEL
LIN {X 0,Y 608.461,Z 127.694,A -85,B 0,C 180,E1 -547.967,E2 -547.967} C_VEL
LIN {X 0,Y 608.425,Z 127.694,A -85,B 0,C 180,E1 -549.415,E2 -549.415} C_VEL
LIN {X 0,Y 607.764,Z 127.78,A -85,B 0,C 180,E1 -549.968,E2 -549.968} C_VEL
LIN {X 0,Y 604.926,Z 128.132,A -85,B 0,C 180,E1 -550.865,E2 -550.865} C_VEL
LIN {X 0,Y 602.515,Z 128.436,A -85,B 0,C 180,E1 -551.586,E2 -551.586} C_VEL
LIN {X 0,Y 601.462,Z 128.562,A -85,B 0,C 180,E1 -552.142,E2 -552.142} C_VEL
LIN {X 0,Y 601.367,Z 128.572,A -85,B 0,C 180,E1 -552.331,E2 -552.331} C_VEL
LIN {X 0,Y 601.366,Z 128.572,A -85,B 0,C 180,E1 -554.898,E2 -554.898} C_VEL
LIN {X 0,Y 601.362,Z 128.579,A -85,B 0,C 180,E1 -557.689,E2 -557.689} C_VEL
LIN {X 0,Y 601.373,Z 128.575,A -85,B 0,C 180,E1 -559.81,E2 -559.81} C_VEL
LIN {X 0,Y 601.378,Z 128.572,A -85,B 0,C 180,E1 -561.96,E2 -561.96} C_VEL
LIN {X 0,Y 601.383,Z 128.579,A -85,B 0,C 180,E1 -564.625,E2 -564.625} C_VEL
LIN {X 0,Y 601.474,Z 142.222,A -85,B 0,C 180,E1 -566.922,E2 -566.922} C_VEL
LIN {X 0,Y 601.428,Z 159.419,A -85,B 0,C 180,E1 -569.773,E2 -569.773} C_VEL
LIN {X 0,Y 601.446,Z 166.076,A -85,B 0,C 180,E1 -570.867,E2 -570.867} C_VEL
LIN {X 0,Y 601.686,Z 169.077,A -85,B 0,C 180,E1 -570.926,E2 -570.926} C_VEL
LIN {X 0,Y 601.589,Z 273.617,A -85,B 0,C 180,E1 -572.196,E2 -572.196} C_VEL
LIN {X 0,Y 601.586,Z 287,A -85,B 0,C 180,E1 -572.506,E2 -572.506} C_VEL
LIN {X 0,Y 601.556,Z 299.98,A -85,B 0,C 180,E1 -572.95,E2 -572.95} C_VEL
LIN {X 0,Y 601.478,Z 311.919,A -85,B 0,C 180,E1 -573.51,E2 -573.51} C_VEL
LIN {X 0,Y 601.471,Z 322.1,A -85,B 0,C 180,E1 -574.115,E2 -574.115} C_VEL
LIN {X 0,Y 601.444,Z 331.87,A -85,B 0,C 180,E1 -574.828,E2 -574.828} C_VEL
LIN {X 0,Y 601.428,Z 340.388,A -85,B 0,C 180,E1 -575.578,E2 -575.578} C_VEL
LIN {X 0,Y 601.384,Z 349.729,A -85,B 0,C 180,E1 -576.584,E2 -576.584} C_VEL
LIN {X 0,Y 601.356,Z 357.507,A -85,B 0,C 180,E1 -577.636,E2 -577.636} C_VEL
LIN {X 0,Y 601.369,Z 364.16,A -85,B 0,C 180,E1 -578.772,E2 -578.772} C_VEL
LIN {X 0,Y 601.351,Z 369.59,A -85,B 0,C 180,E1 -579.999,E2 -579.999} C_VEL
LIN {X 0,Y 601.328,Z 372.528,A -85,B 0,C 180,E1 -580.881,E2 -580.881} C_VEL
LIN {X 0,Y 601.322,Z 374.691,A -85,B 0,C 180,E1 -581.773,E2 -581.773} C_VEL
LIN {X 0,Y 601.34,Z 376.148,A -85,B 0,C 180,E1 -582.676,E2 -582.676} C_VEL
LIN {X 0,Y 601.339,Z 376.898,A -85,B 0,C 180,E1 -583.594,E2 -583.594} C_VEL
LIN {X 0,Y 601.334,Z 376.588,A -85,B 0,C 180,E1 -584.998,E2 -584.998} C_VEL
LIN {X 0,Y 601.339,Z 374.498,A -85,B 0,C 180,E1 -586.407,E2 -586.407} C_VEL
LIN {X 0,Y 601.34,Z 371.879,A -85,B 0,C 180,E1 -587.416,E2 -587.416} C_VEL
LIN {X 0,Y 601.347,Z 368.31,A -85,B 0,C 180,E1 -588.415,E2 -588.415} C_VEL
LIN {X 0,Y 601.347,Z 363.549,A -85,B 0,C 180,E1 -589.434,E2 -589.434} C_VEL
LIN {X 0,Y 601.371,Z 357.39,A -85,B 0,C 180,E1 -590.472,E2 -590.472} C_VEL
LIN {X 0,Y 601.377,Z 349.496,A -85,B 0,C 180,E1 -591.535,E2 -591.535} C_VEL
LIN {X 0,Y 601.431,Z 340.765,A -85,B 0,C 180,E1 -592.476,E2 -592.476} C_VEL
LIN {X 0,Y 601.467,Z 331.17,A -85,B 0,C 180,E1 -593.318,E2 -593.318} C_VEL
LIN {X 0,Y 601.46,Z 320.646,A -85,B 0,C 180,E1 -594.072,E2 -594.072} C_VEL
LIN {X 0,Y 601.5,Z 310.025,A -85,B 0,C 180,E1 -594.681,E2 -594.681} C_VEL
LIN {X 0,Y 601.534,Z 297.64,A -85,B 0,C 180,E1 -595.23,E2 -595.23} C_VEL
LIN {X 0,Y 601.561,Z 285.099,A -85,B 0,C 180,E1 -595.638,E2 -595.638} C_VEL
LIN {X 0,Y 601.601,Z 271.957,A -85,B 0,C 180,E1 -595.922,E2 -595.922} C_VEL
LIN {X 0,Y 601.568,Z 167.233,A -85,B 0,C 180,E1 -597.188,E2 -597.188} C_VEL
LIN {X 0,Y 601.44,Z 166.106,A -85,B 0,C 180,E1 -597.218,E2 -597.218} C_VEL
LIN {X 0,Y 601.461,Z 149.002,A -85,B 0,C 180,E1 -600.039,E2 -600.039} C_VEL
LIN {X 0,Y 601.499,Z 133.551,A -85,B 0,C 180,E1 -602.621,E2 -602.621} C_VEL
LIN {X 0,Y 601.353,Z 128.575,A -85,B 0,C 180,E1 -603.494,E2 -603.494} C_VEL
LIN {X 0,Y 601.388,Z 128.569,A -85,B 0,C 180,E1 -605.857,E2 -605.857} C_VEL
LIN {X 0,Y 601.387,Z 128.575,A -85,B 0,C 180,E1 -608.76,E2 -608.76} C_VEL
LIN {X 0,Y 601.355,Z 128.572,A -85,B 0,C 180,E1 -611.607,E2 -611.607} C_VEL
LIN {X 0,Y 601.385,Z 128.578,A -85,B 0,C 180,E1 -614.408,E2 -614.408} C_VEL
LIN {X 0,Y 601.385,Z 128.577,A -85,B 0,C 180,E1 -616.484,E2 -616.484} C_VEL
LIN {X 0,Y 601.353,Z 128.572,A -85,B 0,C 180,E1 -619.223,E2 -619.223} C_VEL
LIN {X 0,Y 601.424,Z 128.568,A -85,B 0,C 180,E1 -621.939,E2 -621.939} C_VEL
LIN {X 0,Y 601.391,Z 128.571,A -85,B 0,C 180,E1 -624.636,E2 -624.636} C_VEL
LIN {X 0,Y 601.391,Z 128.567,A -85,B 0,C 180,E1 -627.321,E2 -627.321} C_VEL
LIN {X 0,Y 601.44,Z 128.57,A -85,B 0,C 180,E1 -630,E2 -630} C_VEL
LIN {X 0,Y 601.394,Z 128.568,A -85,B 0,C 180,E1 -632.679,E2 -632.679} C_VEL
LIN {X 0,Y 601.385,Z 128.57,A -85,B 0,C 180,E1 -635.364,E2 -635.364} C_VEL
LIN {X 0,Y 601.425,Z 128.571,A -85,B 0,C 180,E1 -638.061,E2 -638.061} C_VEL
LIN {X 0,Y 601.37,Z 128.57,A -85,B 0,C 180,E1 -640.987,E2 -640.987} C_VEL
LIN {X 0,Y 601.388,Z 128.573,A -85,B 0,C 180,E1 -643.516,E2 -643.516} C_VEL
LIN {X 0,Y 601.385,Z 128.57,A -85,B 0,C 180,E1 -646.288,E2 -646.288} C_VEL
LIN {X 0,Y 601.395,Z 128.569,A -85,B 0,C 180,E1 -649.099,E2 -649.099} C_VEL
LIN {X 0,Y 601.372,Z 128.574,A -85,B 0,C 180,E1 -651.961,E2 -651.961} C_VEL
LIN {X 0,Y 601.372,Z 128.571,A -85,B 0,C 180,E1 -654.88,E2 -654.88} C_VEL
LIN {X 0,Y 601.394,Z 128.575,A -85,B 0,C 180,E1 -657.359,E2 -657.359} C_VEL
LIN {X 0,Y 601.366,Z 128.571,A -85,B 0,C 180,E1 -660.167,E2 -660.167} C_VEL
LIN {X 0,Y 601.383,Z 128.57,A -85,B 0,C 180,E1 -662.71,E2 -662.71} C_VEL
LIN {X 0,Y 601.364,Z 128.578,A -85,B 0,C 180,E1 -665.108,E2 -665.108} C_VEL
LIN {X 0,Y 601.424,Z 128.571,A -85,B 0,C 180,E1 -667.419,E2 -667.419} C_VEL
LIN {X 0,Y 601.369,Z 128.57,A -85,B 0,C 180,E1 -669.998,E2 -669.998} C_VEL
LIN {X 0,Y 601.365,Z 128.574,A -85,B 0,C 180,E1 -672.674,E2 -672.674} C_VEL
LIN {X 0,Y 601.392,Z 128.571,A -85,B 0,C 180,E1 -675.479,E2 -675.479} C_VEL
LIN {X 0,Y 601.397,Z 128.568,A -85,B 0,C 180,E1 -678.409,E2 -678.409} C_VEL
LIN {X 0,Y 601.392,Z 128.576,A -85,B 0,C 180,E1 -680.872,E2 -680.872} C_VEL
LIN {X 0,Y 601.38,Z 128.571,A -85,B 0,C 180,E1 -683.416,E2 -683.416} C_VEL
LIN {X 0,Y 601.39,Z 128.568,A -85,B 0,C 180,E1 -686.069,E2 -686.069} C_VEL
LIN {X 0,Y 601.384,Z 128.573,A -85,B 0,C 180,E1 -689.056,E2 -689.056} C_VEL
LIN {X 0,Y 601.38,Z 128.57,A -85,B 0,C 180,E1 -691.371,E2 -691.371} C_VEL
LIN {X 0,Y 601.364,Z 128.57,A -85,B 0,C 180,E1 -693.635,E2 -693.635} C_VEL
LIN {X 0,Y 601.386,Z 128.568,A -85,B 0,C 180,E1 -695.857,E2 -695.857} C_VEL
LIN {X 0,Y 601.386,Z 128.574,A -85,B 0,C 180,E1 -698.76,E2 -698.76} C_VEL
LIN {X 0,Y 601.351,Z 128.572,A -85,B 0,C 180,E1 -701.606,E2 -701.606} C_VEL
LIN {X 0,Y 601.382,Z 128.579,A -85,B 0,C 180,E1 -704.408,E2 -704.408} C_VEL
LIN {X 0,Y 601.382,Z 128.577,A -85,B 0,C 180,E1 -706.484,E2 -706.484} C_VEL
LIN {X 0,Y 601.349,Z 128.572,A -85,B 0,C 180,E1 -709.223,E2 -709.223} C_VEL
LIN {X 0,Y 601.421,Z 128.569,A -85,B 0,C 180,E1 -711.939,E2 -711.939} C_VEL
LIN {X 0,Y 601.388,Z 128.571,A -85,B 0,C 180,E1 -714.636,E2 -714.636} C_VEL
LIN {X 0,Y 601.388,Z 128.568,A -85,B 0,C 180,E1 -717.321,E2 -717.321} C_VEL
LIN {X 0,Y 601.437,Z 128.571,A -85,B 0,C 180,E1 -720,E2 -720} C_VEL
LIN {X 0,Y 601.391,Z 128.568,A -85,B 0,C 180,E1 -722.68,E2 -722.68} C_VEL
LIN {X 0,Y 601.384,Z 128.57,A -85,B 0,C 180,E1 -725.365,E2 -725.365} C_VEL
LIN {X 0,Y 601.422,Z 128.571,A -85,B 0,C 180,E1 -728.061,E2 -728.061} C_VEL
LIN {X 0,Y 601.349,Z 128.572,A -85,B 0,C 180,E1 -730.778,E2 -730.778} C_VEL
LIN {X 0,Y 601.381,Z 128.575,A -85,B 0,C 180,E1 -733.517,E2 -733.517} C_VEL
LIN {X 0,Y 601.385,Z 128.57,A -85,B 0,C 180,E1 -736.289,E2 -736.289} C_VEL
LIN {X 0,Y 601.393,Z 128.569,A -85,B 0,C 180,E1 -739.1,E2 -739.1} C_VEL
LIN {X 0,Y 601.37,Z 128.574,A -85,B 0,C 180,E1 -741.961,E2 -741.961} C_VEL
LIN {X 0,Y 601.369,Z 128.571,A -85,B 0,C 180,E1 -744.88,E2 -744.88} C_VEL
LIN {X 0,Y 601.393,Z 128.576,A -85,B 0,C 180,E1 -747.36,E2 -747.36} C_VEL
LIN {X 0,Y 601.366,Z 128.571,A -85,B 0,C 180,E1 -750.168,E2 -750.168} C_VEL
LIN {X 0,Y 601.381,Z 128.57,A -85,B 0,C 180,E1 -752.71,E2 -752.71} C_VEL
LIN {X 0,Y 601.363,Z 128.578,A -85,B 0,C 180,E1 -755.109,E2 -755.109} C_VEL
LIN {X 0,Y 601.425,Z 128.57,A -85,B 0,C 180,E1 -757.42,E2 -757.42} C_VEL
LIN {X 0,Y 601.371,Z 128.57,A -85,B 0,C 180,E1 -759.999,E2 -759.999} C_VEL
LIN {X 0,Y 601.363,Z 128.574,A -85,B 0,C 180,E1 -762.675,E2 -762.675} C_VEL
LIN {X 0,Y 601.397,Z 128.57,A -85,B 0,C 180,E1 -765.48,E2 -765.48} C_VEL
LIN {X 0,Y 601.397,Z 128.568,A -85,B 0,C 180,E1 -768.41,E2 -768.41} C_VEL
LIN {X 0,Y 601.393,Z 128.577,A -85,B 0,C 180,E1 -770.873,E2 -770.873} C_VEL
LIN {X 0,Y 601.374,Z 128.571,A -85,B 0,C 180,E1 -773.416,E2 -773.416} C_VEL
LIN {X 0,Y 601.396,Z 128.567,A -85,B 0,C 180,E1 -776.07,E2 -776.07} C_VEL
LIN {X 0,Y 601.385,Z 128.573,A -85,B 0,C 180,E1 -779.056,E2 -779.056} C_VEL
LIN {X 0,Y 601.379,Z 128.57,A -85,B 0,C 180,E1 -781.371,E2 -781.371} C_VEL
LIN {X 0,Y 601.364,Z 128.571,A -85,B 0,C 180,E1 -783.635,E2 -783.635} C_VEL
LIN {X 0,Y 601.387,Z 128.569,A -85,B 0,C 180,E1 -785.857,E2 -785.857} C_VEL
LIN {X 0,Y 601.385,Z 128.675,A -85,B 0,C 180,E1 -787.565,E2 -787.565} C_VEL
LIN {X 0,Y 601.618,Z 137.022,A -85,B 0,C 180,E1 -788.769,E2 -788.769} C_VEL
LIN {X 0,Y 601.555,Z 153.826,A -85,B 0,C 180,E1 -791.144,E2 -791.144} C_VEL
LIN {X 0,Y 601.514,Z 173.542,A -85,B 0,C 180,E1 -793.89,E2 -793.89} C_VEL
LIN {X 0,Y 601.445,Z 194.793,A -85,B 0,C 180,E1 -796.807,E2 -796.807} C_VEL
LIN {X 0,Y 601.651,Z 200.515,A -85,B 0,C 180,E1 -796.898,E2 -796.898} C_VEL
LIN {X 0,Y 601.614,Z 302.95,A -85,B 0,C 180,E1 -798.14,E2 -798.14} C_VEL
LIN {X 0,Y 601.56,Z 316.22,A -85,B 0,C 180,E1 -798.438,E2 -798.438} C_VEL
LIN {X 0,Y 601.539,Z 327.945,A -85,B 0,C 180,E1 -798.827,E2 -798.827} C_VEL
LIN {X 0,Y 601.514,Z 338.925,A -85,B 0,C 180,E1 -799.311,E2 -799.311} C_VEL
LIN {X 0,Y 601.474,Z 349.582,A -85,B 0,C 180,E1 -799.906,E2 -799.906} C_VEL
LIN {X 0,Y 601.449,Z 360.477,A -85,B 0,C 180,E1 -800.669,E2 -800.669} C_VEL
LIN {X 0,Y 601.429,Z 371.112,A -85,B 0,C 180,E1 -801.601,E2 -801.601} C_VEL
LIN {X 0,Y 601.418,Z 378.96,A -85,B 0,C 180,E1 -802.446,E2 -802.446} C_VEL
LIN {X 0,Y 601.37,Z 386.225,A -85,B 0,C 180,E1 -803.398,E2 -803.398} C_VEL
LIN {X 0,Y 601.372,Z 391.866,A -85,B 0,C 180,E1 -804.299,E2 -804.299} C_VEL
LIN {X 0,Y 601.336,Z 396.95,A -85,B 0,C 180,E1 -805.307,E2 -805.307} C_VEL
LIN {X 0,Y 601.368,Z 400.896,A -85,B 0,C 180,E1 -806.315,E2 -806.315} C_VEL
LIN {X 0,Y 601.325,Z 403.809,A -85,B 0,C 180,E1 -807.32,E2 -807.32} C_VEL
LIN {X 0,Y 601.343,Z 405.202,A -85,B 0,C 180,E1 -807.991,E2 -807.991} C_VEL
LIN {X 0,Y 601.339,Z 406.784,A -85,B 0,C 180,E1 -809.33,E2 -809.33} C_VEL
LIN {X 0,Y 601.335,Z 407,A -85,B 0,C 180,E1 -810,E2 -810} C_VEL
LIN {X 0,Y 601.347,Z 406.185,A -85,B 0,C 180,E1 -811.339,E2 -811.339} C_VEL
LIN {X 0,Y 601.343,Z 405.202,A -85,B 0,C 180,E1 -812.009,E2 -812.009} C_VEL
LIN {X 0,Y 601.325,Z 403.81,A -85,B 0,C 180,E1 -812.679,E2 -812.679} C_VEL
LIN {X 0,Y 601.368,Z 400.897,A -85,B 0,C 180,E1 -813.685,E2 -813.685} C_VEL
LIN {X 0,Y 601.336,Z 396.95,A -85,B 0,C 180,E1 -814.692,E2 -814.692} C_VEL
LIN {X 0,Y 601.373,Z 390.878,A -85,B 0,C 180,E1 -815.869,E2 -815.869} C_VEL
LIN {X 0,Y 601.382,Z 384.237,A -85,B 0,C 180,E1 -816.88,E2 -816.88} C_VEL
LIN {X 0,Y 601.4,Z 375.991,A -85,B 0,C 180,E1 -817.892,E2 -817.892} C_VEL
LIN {X 0,Y 601.436,Z 367.54,A -85,B 0,C 180,E1 -818.737,E2 -818.737} C_VEL
LIN {X 0,Y 601.449,Z 357.096,A -85,B 0,C 180,E1 -819.585,E2 -819.585} C_VEL
LIN {X 0,Y 601.467,Z 346.762,A -85,B 0,C 180,E1 -820.264,E2 -820.264} C_VEL
LIN {X 0,Y 601.537,Z 334.601,A -85,B 0,C 180,E1 -820.896,E2 -820.896} C_VEL
LIN {X 0,Y 601.555,Z 322.225,A -85,B 0,C 180,E1 -821.378,E2 -821.378} C_VEL
LIN {X 0,Y 601.583,Z 309.449,A -85,B 0,C 180,E1 -821.733,E2 -821.733} C_VEL
LIN {X 0,Y 601.62,Z 297.106,A -85,B 0,C 180,E1 -821.946,E2 -821.946} C_VEL
LIN {X 0,Y 601.551,Z 195.838,A -85,B 0,C 180,E1 -823.16,E2 -823.16} C_VEL
LIN {X 0,Y 601.442,Z 194.637,A -85,B 0,C 180,E1 -823.214,E2 -823.214} C_VEL
LIN {X 0,Y 601.515,Z 173.544,A -85,B 0,C 180,E1 -826.11,E2 -826.11} C_VEL
LIN {X 0,Y 601.596,Z 152.135,A -85,B 0,C 180,E1 -829.093,E2 -829.093} C_VEL
LIN {X 0,Y 601.625,Z 131.986,A -85,B 0,C 180,E1 -831.951,E2 -831.951} C_VEL
LIN {X 0,Y 601.371,Z 128.574,A -85,B 0,C 180,E1 -832.461,E2 -832.461} C_VEL
LIN {X 0,Y 601.37,Z 128.573,A -85,B 0,C 180,E1 -834.88,E2 -834.88} C_VEL
LIN {X 0,Y 601.395,Z 128.578,A -85,B 0,C 180,E1 -837.358,E2 -837.358} C_VEL
LIN {X 0,Y 601.368,Z 128.571,A -85,B 0,C 180,E1 -840.167,E2 -840.167} C_VEL
LIN {X 0,Y 601.381,Z 128.571,A -85,B 0,C 180,E1 -842.709,E2 -842.709} C_VEL
LIN {X 0,Y 601.364,Z 128.58,A -85,B 0,C 180,E1 -845.107,E2 -845.107} C_VEL
LIN {X 0,Y 601.425,Z 128.569,A -85,B 0,C 180,E1 -847.419,E2 -847.419} C_VEL
LIN {X 0,Y 601.37,Z 128.57,A -85,B 0,C 180,E1 -849.997,E2 -849.997} C_VEL
LIN {X 0,Y 601.365,Z 128.576,A -85,B 0,C 180,E1 -852.673,E2 -852.673} C_VEL
LIN {X 0,Y 601.395,Z 128.569,A -85,B 0,C 180,E1 -855.479,E2 -855.479} C_VEL
LIN {X 0,Y 601.397,Z 128.569,A -85,B 0,C 180,E1 -858.409,E2 -858.409} C_VEL
LIN {X 0,Y 601.391,Z 128.577,A -85,B 0,C 180,E1 -860.872,E2 -860.872} C_VEL
LIN {X 0,Y 601.375,Z 128.57,A -85,B 0,C 180,E1 -863.415,E2 -863.415} C_VEL
LIN {X 0,Y 601.391,Z 128.569,A -85,B 0,C 180,E1 -866.069,E2 -866.069} C_VEL
LIN {X 0,Y 601.382,Z 128.572,A -85,B 0,C 180,E1 -869.056,E2 -869.056} C_VEL
LIN {X 0,Y 601.377,Z 128.57,A -85,B 0,C 180,E1 -871.37,E2 -871.37} C_VEL
LIN {X 0,Y 601.386,Z 128.572,A -85,B 0,C 180,E1 -874.136,E2 -874.136} C_VEL
LIN {X 0,Y 601.366,Z 128.579,A -85,B 0,C 180,E1 -876.587,E2 -876.587} C_VEL
LIN {X 0,Y 601.379,Z 128.569,A -85,B 0,C 180,E1 -879.476,E2 -879.476} C_VEL
LIN {X 0,Y 601.352,Z 128.572,A -85,B 0,C 180,E1 -881.606,E2 -881.606} C_VEL
LIN {X 0,Y 601.381,Z 128.577,A -85,B 0,C 180,E1 -884.408,E2 -884.408} C_VEL
LIN {X 0,Y 601.38,Z 128.575,A -85,B 0,C 180,E1 -886.483,E2 -886.483} C_VEL
LIN {X 0,Y 601.349,Z 128.572,A -85,B 0,C 180,E1 -889.222,E2 -889.222} C_VEL
LIN {X 0,Y 601.42,Z 128.571,A -85,B 0,C 180,E1 -891.939,E2 -891.939} C_VEL
LIN {X 0,Y 601.383,Z 128.57,A -85,B 0,C 180,E1 -894.635,E2 -894.635} C_VEL
LIN {X 0,Y 601.389,Z 128.569,A -85,B 0,C 180,E1 -897.32,E2 -897.32} C_VEL
LIN {X 0,Y 601.436,Z 128.571,A -85,B 0,C 180,E1 -900,E2 -900} C_VEL
LIN {X 0,Y 601.387,Z 128.568,A -85,B 0,C 180,E1 -902.679,E2 -902.679} C_VEL
LIN {X 0,Y 601.387,Z 128.571,A -85,B 0,C 180,E1 -905.364,E2 -905.364} C_VEL
LIN {X 0,Y 601.42,Z 128.569,A -85,B 0,C 180,E1 -908.061,E2 -908.061} C_VEL
LIN {X 0,Y 601.369,Z 128.571,A -85,B 0,C 180,E1 -910.989,E2 -910.989} C_VEL
LIN {X 0,Y 601.367,Z 128.572,A -85,B 0,C 180,E1 -912.331,E2 -912.331} C_VEL
LIN {X 0,Y 600.676,Z 128.658,A -85,B 0,C 180,E1 -912.89,E2 -912.89} C_VEL
LIN {X 0,Y 597.822,Z 129.02,A -85,B 0,C 180,E1 -913.798,E2 -913.798} C_VEL
LIN {X 0,Y 595.427,Z 129.316,A -85,B 0,C 180,E1 -914.528,E2 -914.528} C_VEL
LIN {X 0,Y 594.399,Z 129.441,A -85,B 0,C 180,E1 -915.092,E2 -915.092} C_VEL
LIN {X 0,Y 594.315,Z 129.452,A -85,B 0,C 180,E1 -915.283,E2 -915.283} C_VEL
LIN {X 0,Y 594.31,Z 129.454,A -85,B 0,C 180,E1 -917.906,E2 -917.906} C_VEL
LIN {X 0,Y 594.361,Z 129.445,A -85,B 0,C 180,E1 -920.777,E2 -920.777} C_VEL
LIN {X 0,Y 594.33,Z 129.454,A -85,B 0,C 180,E1 -923.706,E2 -923.706} C_VEL
LIN {X 0,Y 594.342,Z 129.484,A -85,B 0,C 180,E1 -924.541,E2 -924.541} C_VEL
LIN {X 0,Y 594.491,Z 139.939,A -85,B 0,C 180,E1 -926.328,E2 -926.328} C_VEL
LIN {X 0,Y 594.437,Z 156.951,A -85,B 0,C 180,E1 -929.189,E2 -929.189} C_VEL
LIN {X 0,Y 594.401,Z 166.412,A -85,B 0,C 180,E1 -930.73,E2 -930.73} C_VEL
LIN {X 0,Y 594.771,Z 171.068,A -85,B 0,C 180,E1 -930.795,E2 -930.795} C_VEL
LIN {X 0,Y 594.668,Z 273.13,A -85,B 0,C 180,E1 -932.047,E2 -932.047} C_VEL
LIN {X 0,Y 594.606,Z 286.154,A -85,B 0,C 180,E1 -932.345,E2 -932.345} C_VEL
LIN {X 0,Y 594.576,Z 297.848,A -85,B 0,C 180,E1 -932.736,E2 -932.736} C_VEL
LIN {X 0,Y 594.504,Z 309.272,A -85,B 0,C 180,E1 -933.245,E2 -933.245} C_VEL
LIN {X 0,Y 594.469,Z 320.623,A -85,B 0,C 180,E1 -933.898,E2 -933.898} C_VEL
LIN {X 0,Y 594.394,Z 331.417,A -85,B 0,C 180,E1 -934.682,E2 -934.682} C_VEL
LIN {X 0,Y 594.388,Z 340.721,A -85,B 0,C 180,E1 -935.51,E2 -935.51} C_VEL
LIN {X 0,Y 594.331,Z 349.594,A -85,B 0,C 180,E1 -936.478,E2 -936.478} C_VEL
LIN {X 0,Y 594.271,Z 357.745,A -85,B 0,C 180,E1 -937.595,E2 -937.595} C_VEL
LIN {X 0,Y 594.299,Z 364.075,A -85,B 0,C 180,E1 -938.695,E2 -938.695} C_VEL
LIN {X 0,Y 594.254,Z 368.868,A -85,B 0,C 180,E1 -939.761,E2 -939.761} C_VEL
LIN {X 0,Y 594.228,Z 372.412,A -85,B 0,C 180,E1 -940.806,E2 -940.806} C_VEL
LIN {X 0,Y 594.245,Z 374.873,A -85,B 0,C 180,E1 -941.835,E2 -941.835} C_VEL
LIN {X 0,Y 594.245,Z 376.355,A -85,B 0,C 180,E1 -942.841,E2 -942.841} C_VEL
LIN {X 0,Y 594.224,Z 376.959,A -85,B 0,C 180,E1 -944.251,E2 -944.251} C_VEL
LIN {X 0,Y 594.241,Z 376.408,A -85,B 0,C 180,E1 -945.203,E2 -945.203} C_VEL
LIN {X 0,Y 594.231,Z 375.04,A -85,B 0,C 180,E1 -946.174,E2 -946.174} C_VEL
LIN {X 0,Y 594.249,Z 372.766,A -85,B 0,C 180,E1 -947.16,E2 -947.16} C_VEL
LIN {X 0,Y 594.245,Z 368.062,A -85,B 0,C 180,E1 -948.525,E2 -948.525} C_VEL
LIN {X 0,Y 594.284,Z 362.779,A -85,B 0,C 180,E1 -949.642,E2 -949.642} C_VEL
LIN {X 0,Y 594.309,Z 356.042,A -85,B 0,C 180,E1 -950.754,E2 -950.754} C_VEL
LIN {X 0,Y 594.327,Z 349.022,A -85,B 0,C 180,E1 -951.682,E2 -951.682} C_VEL
LIN {X 0,Y 594.388,Z 341.192,A -85,B 0,C 180,E1 -952.535,E2 -952.535} C_VEL
LIN {X 0,Y 594.439,Z 331.411,A -85,B 0,C 180,E1 -953.408,E2 -953.408} C_VEL
LIN {X 0,Y 594.461,Z 320.758,A -85,B 0,C 180,E1 -954.183,E2 -954.183} C_VEL
LIN {X 0,Y 594.501,Z 308.938,A -85,B 0,C 180,E1 -954.861,E2 -954.861} C_VEL
LIN {X 0,Y 594.562,Z 297.149,A -85,B 0,C 180,E1 -955.381,E2 -955.381} C_VEL
LIN {X 0,Y 594.637,Z 284.579,A -85,B 0,C 180,E1 -955.788,E2 -955.788} C_VEL
LIN {X 0,Y 594.662,Z 272.384,A -85,B 0,C 180,E1 -956.056,E2 -956.056} C_VEL
LIN {X 0,Y 594.737,Z 168.663,A -85,B 0,C 180,E1 -957.325,E2 -957.325} C_VEL
LIN {X 0,Y 594.373,Z 166.108,A -85,B 0,C 180,E1 -957.378,E2 -957.378} C_VEL
LIN {X 0,Y 594.45,Z 149.031,A -85,B 0,C 180,E1 -960.228,E2 -960.228} C_VEL
LIN {X 0,Y 594.515,Z 133.084,A -85,B 0,C 180,E1 -962.928,E2 -962.928} C_VEL
LIN {X 0,Y 594.345,Z 129.449,A -85,B 0,C 180,E1 -963.583,E2 -963.583} C_VEL
LIN {X 0,Y 594.336,Z 129.452,A -85,B 0,C 180,E1 -966.294,E2 -966.294} C_VEL
LIN {X 0,Y 594.365,Z 129.444,A -85,B 0,C 180,E1 -969.223,E2 -969.223} C_VEL
LIN {X 0,Y 594.316,Z 129.452,A -85,B 0,C 180,E1 -972.094,E2 -972.094} C_VEL
LIN {X 0,Y 594.328,Z 129.45,A -85,B 0,C 180,E1 -974.921,E2 -974.921} C_VEL
LIN {X 0,Y 594.339,Z 129.447,A -85,B 0,C 180,E1 -977.711,E2 -977.711} C_VEL
LIN {X 0,Y 594.34,Z 129.453,A -85,B 0,C 180,E1 -980.471,E2 -980.471} C_VEL
LIN {X 0,Y 594.335,Z 129.446,A -85,B 0,C 180,E1 -983.209,E2 -983.209} C_VEL
LIN {X 0,Y 594.344,Z 129.451,A -85,B 0,C 180,E1 -985.932,E2 -985.932} C_VEL
LIN {X 0,Y 594.337,Z 129.448,A -85,B 0,C 180,E1 -988.645,E2 -988.645} C_VEL
LIN {X 0,Y 594.319,Z 129.45,A -85,B 0,C 180,E1 -990.678,E2 -990.678} C_VEL
LIN {X 0,Y 594.362,Z 129.444,A -85,B 0,C 180,E1 -992.711,E2 -992.711} C_VEL
LIN {X 0,Y 594.355,Z 129.446,A -85,B 0,C 180,E1 -995.428,E2 -995.428} C_VEL
LIN {X 0,Y 594.367,Z 129.448,A -85,B 0,C 180,E1 -998.157,E2 -998.157} C_VEL
LIN {X 0,Y 594.327,Z 129.448,A -85,B 0,C 180,E1 -1001.044,E2 -1001.044} C_VEL
LIN {X 0,Y 594.355,Z 129.452,A -85,B 0,C 180,E1 -1003.679,E2 -1003.679} C_VEL
LIN {X 0,Y 594.314,Z 129.449,A -85,B 0,C 180,E1 -1006.694,E2 -1006.694} C_VEL
LIN {X 0,Y 594.347,Z 129.45,A -85,B 0,C 180,E1 -1009.335,E2 -1009.335} C_VEL
LIN {X 0,Y 594.339,Z 129.454,A -85,B 0,C 180,E1 -1011.504,E2 -1011.504} C_VEL
LIN {X 0,Y 594.336,Z 129.446,A -85,B 0,C 180,E1 -1014.448,E2 -1014.448} C_VEL
LIN {X 0,Y 594.348,Z 129.445,A -85,B 0,C 180,E1 -1016.701,E2 -1016.701} C_VEL
LIN {X 0,Y 594.331,Z 129.451,A -85,B 0,C 180,E1 -1019.778,E2 -1019.778} C_VEL
LIN {X 0,Y 594.33,Z 129.447,A -85,B 0,C 180,E1 -1022.149,E2 -1022.149} C_VEL
LIN {X 0,Y 594.348,Z 129.445,A -85,B 0,C 180,E1 -1024.582,E2 -1024.582} C_VEL
LIN {X 0,Y 594.37,Z 129.446,A -85,B 0,C 180,E1 -1027.606,E2 -1027.606} C_VEL
LIN {X 0,Y 594.333,Z 129.448,A -85,B 0,C 180,E1 -1030.569,E2 -1030.569} C_VEL
LIN {X 0,Y 594.335,Z 129.453,A -85,B 0,C 180,E1 -1033.302,E2 -1033.302} C_VEL
LIN {X 0,Y 594.334,Z 129.446,A -85,B 0,C 180,E1 -1036.163,E2 -1036.163} C_VEL
LIN {X 0,Y 594.353,Z 129.451,A -85,B 0,C 180,E1 -1039.18,E2 -1039.18} C_VEL
LIN {X 0,Y 594.34,Z 129.446,A -85,B 0,C 180,E1 -1042.056,E2 -1042.056} C_VEL
LIN {X 0,Y 594.307,Z 129.457,A -85,B 0,C 180,E1 -1044.682,E2 -1044.682} C_VEL
LIN {X 0,Y 594.361,Z 129.448,A -85,B 0,C 180,E1 -1047.09,E2 -1047.09} C_VEL
LIN {X 0,Y 594.338,Z 129.446,A -85,B 0,C 180,E1 -1049.679,E2 -1049.679} C_VEL
LIN {X 0,Y 594.351,Z 129.452,A -85,B 0,C 180,E1 -1052.538,E2 -1052.538} C_VEL
LIN {X 0,Y 594.344,Z 129.452,A -85,B 0,C 180,E1 -1054.806,E2 -1054.806} C_VEL
LIN {X 0,Y 594.299,Z 129.452,A -85,B 0,C 180,E1 -1057.278,E2 -1057.278} C_VEL
LIN {X 0,Y 594.338,Z 129.448,A -85,B 0,C 180,E1 -1059.945,E2 -1059.945} C_VEL
LIN {X 0,Y 594.315,Z 129.453,A -85,B 0,C 180,E1 -1062.805,E2 -1062.805} C_VEL
LIN {X 0,Y 594.342,Z 129.446,A -85,B 0,C 180,E1 -1065.622,E2 -1065.622} C_VEL
LIN {X 0,Y 594.362,Z 129.452,A -85,B 0,C 180,E1 -1068.404,E2 -1068.404} C_VEL
LIN {X 0,Y 594.318,Z 129.448,A -85,B 0,C 180,E1 -1071.157,E2 -1071.157} C_VEL
LIN {X 0,Y 594.354,Z 129.449,A -85,B 0,C 180,E1 -1073.891,E2 -1073.891} C_VEL
LIN {X 0,Y 594.312,Z 129.452,A -85,B 0,C 180,E1 -1076.611,E2 -1076.611} C_VEL
LIN {X 0,Y 594.334,Z 129.448,A -85,B 0,C 180,E1 -1078.645,E2 -1078.645} C_VEL
LIN {X 0,Y 594.316,Z 129.45,A -85,B 0,C 180,E1 -1080.678,E2 -1080.678} C_VEL
LIN {X 0,Y 594.359,Z 129.444,A -85,B 0,C 180,E1 -1082.711,E2 -1082.711} C_VEL
LIN {X 0,Y 594.354,Z 129.446,A -85,B 0,C 180,E1 -1085.428,E2 -1085.428} C_VEL
LIN {X 0,Y 594.364,Z 129.448,A -85,B 0,C 180,E1 -1088.158,E2 -1088.158} C_VEL
LIN {X 0,Y 594.339,Z 129.446,A -85,B 0,C 180,E1 -1091.052,E2 -1091.052} C_VEL
LIN {X 0,Y 594.349,Z 129.454,A -85,B 0,C 180,E1 -1093.68,E2 -1093.68} C_VEL
LIN {X 0,Y 594.313,Z 129.449,A -85,B 0,C 180,E1 -1096.695,E2 -1096.695} C_VEL
LIN {X 0,Y 594.345,Z 129.45,A -85,B 0,C 180,E1 -1099.335,E2 -1099.335} C_VEL
LIN {X 0,Y 594.338,Z 129.455,A -85,B 0,C 180,E1 -1101.505,E2 -1101.505} C_VEL
LIN {X 0,Y 594.335,Z 129.446,A -85,B 0,C 180,E1 -1104.449,E2 -1104.449} C_VEL
LIN {X 0,Y 594.346,Z 129.445,A -85,B 0,C 180,E1 -1106.702,E2 -1106.702} C_VEL
LIN {X 0,Y 594.329,Z 129.451,A -85,B 0,C 180,E1 -1109.779,E2 -1109.779} C_VEL
LIN {X 0,Y 594.329,Z 129.447,A -85,B 0,C 180,E1 -1112.15,E2 -1112.15} C_VEL
LIN {X 0,Y 594.348,Z 129.445,A -85,B 0,C 180,E1 -1114.582,E2 -1114.582} C_VEL
LIN {X 0,Y 594.371,Z 129.446,A -85,B 0,C 180,E1 -1117.607,E2 -1117.607} C_VEL
LIN {X 0,Y 594.335,Z 129.448,A -85,B 0,C 180,E1 -1120.57,E2 -1120.57} C_VEL
LIN {X 0,Y 594.337,Z 129.453,A -85,B 0,C 180,E1 -1123.303,E2 -1123.303} C_VEL
LIN {X 0,Y 594.338,Z 129.446,A -85,B 0,C 180,E1 -1126.164,E2 -1126.164} C_VEL
LIN {X 0,Y 594.355,Z 129.45,A -85,B 0,C 180,E1 -1129.181,E2 -1129.181} C_VEL
LIN {X 0,Y 594.341,Z 129.446,A -85,B 0,C 180,E1 -1132.056,E2 -1132.056} C_VEL
LIN {X 0,Y 594.303,Z 129.458,A -85,B 0,C 180,E1 -1134.683,E2 -1134.683} C_VEL
LIN {X 0,Y 594.337,Z 129.451,A -85,B 0,C 180,E1 -1137.095,E2 -1137.095} C_VEL
LIN {X 0,Y 594.343,Z 129.445,A -85,B 0,C 180,E1 -1139.68,E2 -1139.68} C_VEL
LIN {X 0,Y 594.338,Z 129.454,A -85,B 0,C 180,E1 -1142.538,E2 -1142.538} C_VEL
LIN {X 0,Y 594.326,Z 129.455,A -85,B 0,C 180,E1 -1144.805,E2 -1144.805} C_VEL
LIN {X 0,Y 594.343,Z 129.618,A -85,B 0,C 180,E1 -1147.422,E2 -1147.422} C_VEL
LIN {X 0,Y 594.732,Z 135.763,A -85,B 0,C 180,E1 -1148.329,E2 -1148.329} C_VEL
LIN {X 0,Y 594.596,Z 155.313,A -85,B 0,C 180,E1 -1151.126,E2 -1151.126} C_VEL
LIN {X 0,Y 594.514,Z 176.061,A -85,B 0,C 180,E1 -1154.047,E2 -1154.047} C_VEL
LIN {X 0,Y 594.461,Z 195.149,A -85,B 0,C 180,E1 -1156.671,E2 -1156.671} C_VEL
LIN {X 0,Y 594.73,Z 205.881,A -85,B 0,C 180,E1 -1156.808,E2 -1156.808} C_VEL
LIN {X 0,Y 594.666,Z 302.95,A -85,B 0,C 180,E1 -1157.999,E2 -1157.999} C_VEL
LIN {X 0,Y 594.601,Z 316.221,A -85,B 0,C 180,E1 -1158.3,E2 -1158.3} C_VEL
LIN {X 0,Y 594.572,Z 328.57,A -85,B 0,C 180,E1 -1158.718,E2 -1158.718} C_VEL
LIN {X 0,Y 594.536,Z 340.632,A -85,B 0,C 180,E1 -1159.27,E2 -1159.27} C_VEL
LIN {X 0,Y 594.477,Z 352.202,A -85,B 0,C 180,E1 -1159.958,E2 -1159.958} C_VEL
LIN {X 0,Y 594.414,Z 362.598,A -85,B 0,C 180,E1 -1160.73,E2 -1160.73} C_VEL
LIN {X 0,Y 594.383,Z 371.112,A -85,B 0,C 180,E1 -1161.501,E2 -1161.501} C_VEL
LIN {X 0,Y 594.347,Z 378.96,A -85,B 0,C 180,E1 -1162.355,E2 -1162.355} C_VEL
LIN {X 0,Y 594.283,Z 386.814,A -85,B 0,C 180,E1 -1163.408,E2 -1163.408} C_VEL
LIN {X 0,Y 594.289,Z 393.68,A -85,B 0,C 180,E1 -1164.571,E2 -1164.571} C_VEL
LIN {X 0,Y 594.27,Z 398.371,A -85,B 0,C 180,E1 -1165.591,E2 -1165.591} C_VEL
LIN {X 0,Y 594.267,Z 401.956,A -85,B 0,C 180,E1 -1166.61,E2 -1166.61} C_VEL
LIN {X 0,Y 594.226,Z 403.809,A -85,B 0,C 180,E1 -1167.288,E2 -1167.288} C_VEL
LIN {X 0,Y 594.242,Z 405.2,A -85,B 0,C 180,E1 -1167.967,E2 -1167.967} C_VEL
LIN {X 0,Y 594.239,Z 406.784,A -85,B 0,C 180,E1 -1169.322,E2 -1169.322} C_VEL
LIN {X 0,Y 594.236,Z 407,A -85,B 0,C 180,E1 -1170,E2 -1170} C_VEL
LIN {X 0,Y 594.247,Z 406.185,A -85,B 0,C 180,E1 -1171.355,E2 -1171.355} C_VEL
LIN {X 0,Y 594.242,Z 405.201,A -85,B 0,C 180,E1 -1172.033,E2 -1172.033} C_VEL
LIN {X 0,Y 594.226,Z 403.81,A -85,B 0,C 180,E1 -1172.711,E2 -1172.711} C_VEL
LIN {X 0,Y 594.289,Z 400.897,A -85,B 0,C 180,E1 -1173.729,E2 -1173.729} C_VEL
LIN {X 0,Y 594.241,Z 396.95,A -85,B 0,C 180,E1 -1174.749,E2 -1174.749} C_VEL
LIN {X 0,Y 594.305,Z 390.879,A -85,B 0,C 180,E1 -1175.939,E2 -1175.939} C_VEL
LIN {X 0,Y 594.308,Z 384.238,A -85,B 0,C 180,E1 -1176.962,E2 -1176.962} C_VEL
LIN {X 0,Y 594.359,Z 375.992,A -85,B 0,C 180,E1 -1177.986,E2 -1177.986} C_VEL
LIN {X 0,Y 594.382,Z 367.54,A -85,B 0,C 180,E1 -1178.842,E2 -1178.842} C_VEL
LIN {X 0,Y 594.432,Z 357.098,A -85,B 0,C 180,E1 -1179.699,E2 -1179.699} C_VEL
LIN {X 0,Y 594.481,Z 346.762,A -85,B 0,C 180,E1 -1180.386,E2 -1180.386} C_VEL
LIN {X 0,Y 594.558,Z 335.727,A -85,B 0,C 180,E1 -1180.973,E2 -1180.973} C_VEL
LIN {X 0,Y 594.579,Z 323.719,A -85,B 0,C 180,E1 -1181.464,E2 -1181.464} C_VEL
LIN {X 0,Y 594.624,Z 310.362,A -85,B 0,C 180,E1 -1181.85,E2 -1181.85} C_VEL
LIN {X 0,Y 594.699,Z 297.106,A -85,B 0,C 180,E1 -1182.087,E2 -1182.087} C_VEL
LIN {X 0,Y 594.703,Z 196.956,A -85,B 0,C 180,E1 -1183.301,E2 -1183.301} C_VEL
LIN {X 0,Y 594.422,Z 194.795,A -85,B 0,C 180,E1 -1183.351,E2 -1183.351} C_VEL
LIN {X 0,Y 594.523,Z 173.544,A -85,B 0,C 180,E1 -1186.305,E2 -1186.305} C_VEL
LIN {X 0,Y 594.63,Z 153.726,A -85,B 0,C 180,E1 -1189.099,E2 -1189.099} C_VEL
LIN {X 0,Y 594.704,Z 133.246,A -85,B 0,C 180,E1 -1192.037,E2 -1192.037} C_VEL
LIN {X 0,Y 594.303,Z 129.455,A -85,B 0,C 180,E1 -1192.612,E2 -1192.612} C_VEL
LIN {X 0,Y 594.325,Z 129.455,A -85,B 0,C 180,E1 -1195.195,E2 -1195.195} C_VEL
LIN {X 0,Y 594.342,Z 129.453,A -85,B 0,C 180,E1 -1197.518,E2 -1197.518} C_VEL
LIN {X 0,Y 594.343,Z 129.446,A -85,B 0,C 180,E1 -1200.32,E2 -1200.32} C_VEL
LIN {X 0,Y 594.338,Z 129.452,A -85,B 0,C 180,E1 -1202.952,E2 -1202.952} C_VEL
LIN {X 0,Y 594.299,Z 129.457,A -85,B 0,C 180,E1 -1205.412,E2 -1205.412} C_VEL
LIN {X 0,Y 594.339,Z 129.446,A -85,B 0,C 180,E1 -1207.943,E2 -1207.943} C_VEL
LIN {X 0,Y 594.354,Z 129.451,A -85,B 0,C 180,E1 -1210.819,E2 -1210.819} C_VEL
LIN {X 0,Y 594.336,Z 129.447,A -85,B 0,C 180,E1 -1213.836,E2 -1213.836} C_VEL
LIN {X 0,Y 594.335,Z 129.453,A -85,B 0,C 180,E1 -1216.697,E2 -1216.697} C_VEL
LIN {X 0,Y 594.333,Z 129.448,A -85,B 0,C 180,E1 -1219.43,E2 -1219.43} C_VEL
LIN {X 0,Y 594.369,Z 129.446,A -85,B 0,C 180,E1 -1222.393,E2 -1222.393} C_VEL
LIN {X 0,Y 594.347,Z 129.446,A -85,B 0,C 180,E1 -1225.418,E2 -1225.418} C_VEL
LIN {X 0,Y 594.328,Z 129.447,A -85,B 0,C 180,E1 -1227.85,E2 -1227.85} C_VEL
LIN {X 0,Y 594.327,Z 129.451,A -85,B 0,C 180,E1 -1230.221,E2 -1230.221} C_VEL
LIN {X 0,Y 594.345,Z 129.445,A -85,B 0,C 180,E1 -1233.298,E2 -1233.298} C_VEL
LIN {X 0,Y 594.324,Z 129.448,A -85,B 0,C 180,E1 -1235.578,E2 -1235.578} C_VEL
LIN {X 0,Y 594.337,Z 129.456,A -85,B 0,C 180,E1 -1238.495,E2 -1238.495} C_VEL
LIN {X 0,Y 594.331,Z 129.446,A -85,B 0,C 180,E1 -1241.381,E2 -1241.381} C_VEL
LIN {X 0,Y 594.328,Z 129.456,A -85,B 0,C 180,E1 -1244.218,E2 -1244.218} C_VEL
LIN {X 0,Y 594.347,Z 129.454,A -85,B 0,C 180,E1 -1246.32,E2 -1246.32} C_VEL
LIN {X 0,Y 594.315,Z 129.449,A -85,B 0,C 180,E1 -1249.093,E2 -1249.093} C_VEL
LIN {X 0,Y 594.362,Z 129.448,A -85,B 0,C 180,E1 -1251.842,E2 -1251.842} C_VEL
LIN {X 0,Y 594.353,Z 129.446,A -85,B 0,C 180,E1 -1254.572,E2 -1254.572} C_VEL
LIN {X 0,Y 594.357,Z 129.444,A -85,B 0,C 180,E1 -1257.289,E2 -1257.289} C_VEL
LIN {X 0,Y 594.404,Z 129.447,A -85,B 0,C 180,E1 -1260,E2 -1260} C_VEL
LIN {X 0,Y 594.356,Z 129.444,A -85,B 0,C 180,E1 -1262.711,E2 -1262.711} C_VEL
LIN {X 0,Y 594.356,Z 129.448,A -85,B 0,C 180,E1 -1265.428,E2 -1265.428} C_VEL
LIN {X 0,Y 594.362,Z 129.447,A -85,B 0,C 180,E1 -1268.157,E2 -1268.157} C_VEL
LIN {X 0,Y 594.335,Z 129.448,A -85,B 0,C 180,E1 -1271.051,E2 -1271.051} C_VEL
LIN {X 0,Y 594.347,Z 129.455,A -85,B 0,C 180,E1 -1273.679,E2 -1273.679} C_VEL
LIN {X 0,Y 594.315,Z 129.452,A -85,B 0,C 180,E1 -1275.283,E2 -1275.283} C_VEL
LIN {X 0,Y 593.644,Z 129.54,A -85,B 0,C 180,E1 -1275.848,E2 -1275.848} C_VEL
LIN {X 0,Y 590.777,Z 129.896,A -85,B 0,C 180,E1 -1276.766,E2 -1276.766} C_VEL
LIN {X 0,Y 588.365,Z 130.2,A -85,B 0,C 180,E1 -1277.504,E2 -1277.504} C_VEL
LIN {X 0,Y 587.341,Z 130.321,A -85,B 0,C 180,E1 -1278.074,E2 -1278.074} C_VEL
LIN {X 0,Y 587.264,Z 130.328,A -85,B 0,C 180,E1 -1278.267,E2 -1278.267} C_VEL
LIN {X 0,Y 587.305,Z 130.326,A -85,B 0,C 180,E1 -1281.038,E2 -1281.038} C_VEL
LIN {X 0,Y 587.27,Z 130.33,A -85,B 0,C 180,E1 -1284.009,E2 -1284.009} C_VEL
LIN {X 0,Y 587.302,Z 130.343,A -85,B 0,C 180,E1 -1284.447,E2 -1284.447} C_VEL
LIN {X 0,Y 587.52,Z 137.447,A -85,B 0,C 180,E1 -1285.682,E2 -1285.682} C_VEL
LIN {X 0,Y 587.406,Z 154.503,A -85,B 0,C 180,E1 -1288.592,E2 -1288.592} C_VEL
LIN {X 0,Y 587.344,Z 166.225,A -85,B 0,C 180,E1 -1290.565,E2 -1290.565} C_VEL
LIN {X 0,Y 587.867,Z 171.404,A -85,B 0,C 180,E1 -1290.641,E2 -1290.641} C_VEL
LIN {X 0,Y 587.728,Z 273.446,A -85,B 0,C 180,E1 -1291.909,E2 -1291.909} C_VEL
LIN {X 0,Y 587.661,Z 286.376,A -85,B 0,C 180,E1 -1292.212,E2 -1292.212} C_VEL
LIN {X 0,Y 587.617,Z 299.225,A -85,B 0,C 180,E1 -1292.654,E2 -1292.654} C_VEL
LIN {X 0,Y 587.499,Z 311.167,A -85,B 0,C 180,E1 -1293.215,E2 -1293.215} C_VEL
LIN {X 0,Y 587.445,Z 322.491,A -85,B 0,C 180,E1 -1293.904,E2 -1293.904} C_VEL
LIN {X 0,Y 587.386,Z 332.65,A -85,B 0,C 180,E1 -1294.671,E2 -1294.671} C_VEL
LIN {X 0,Y 587.305,Z 342.08,A -85,B 0,C 180,E1 -1295.54,E2 -1295.54} C_VEL
LIN {X 0,Y 587.27,Z 350.565,A -85,B 0,C 180,E1 -1296.509,E2 -1296.509} C_VEL
LIN {X 0,Y 587.231,Z 356.984,A -85,B 0,C 180,E1 -1297.4,E2 -1297.4} C_VEL
LIN {X 0,Y 587.191,Z 363.353,A -85,B 0,C 180,E1 -1298.49,E2 -1298.49} C_VEL
LIN {X 0,Y 587.167,Z 368.772,A -85,B 0,C 180,E1 -1299.688,E2 -1299.688} C_VEL
LIN {X 0,Y 587.156,Z 372.066,A -85,B 0,C 180,E1 -1300.657,E2 -1300.657} C_VEL
LIN {X 0,Y 587.124,Z 373.496,A -85,B 0,C 180,E1 -1301.175,E2 -1301.175} C_VEL
LIN {X 0,Y 587.156,Z 375.372,A -85,B 0,C 180,E1 -1302.089,E2 -1302.089} C_VEL
LIN {X 0,Y 587.143,Z 376.612,A -85,B 0,C 180,E1 -1303.101,E2 -1303.101} C_VEL
LIN {X 0,Y 587.149,Z 376.994,A -85,B 0,C 180,E1 -1304.096,E2 -1304.096} C_VEL
LIN {X 0,Y 587.163,Z 376.552,A -85,B 0,C 180,E1 -1305.075,E2 -1305.075} C_VEL
LIN {X 0,Y 587.13,Z 375.32,A -85,B 0,C 180,E1 -1306.032,E2 -1306.032} C_VEL
LIN {X 0,Y 587.165,Z 373.326,A -85,B 0,C 180,E1 -1306.981,E2 -1306.981} C_VEL
LIN {X 0,Y 587.186,Z 370.576,A -85,B 0,C 180,E1 -1307.914,E2 -1307.914} C_VEL
LIN {X 0,Y 587.181,Z 366.554,A -85,B 0,C 180,E1 -1308.942,E2 -1308.942} C_VEL
LIN {X 0,Y 587.207,Z 361.244,A -85,B 0,C 180,E1 -1309.994,E2 -1309.994} C_VEL
LIN {X 0,Y 587.262,Z 354.405,A -85,B 0,C 180,E1 -1311.066,E2 -1311.066} C_VEL
LIN {X 0,Y 587.286,Z 346.674,A -85,B 0,C 180,E1 -1312.046,E2 -1312.046} C_VEL
LIN {X 0,Y 587.349,Z 338.144,A -85,B 0,C 180,E1 -1312.932,E2 -1312.932} C_VEL
LIN {X 0,Y 587.413,Z 328.045,A -85,B 0,C 180,E1 -1313.791,E2 -1313.791} C_VEL
LIN {X 0,Y 587.453,Z 316.11,A -85,B 0,C 180,E1 -1314.595,E2 -1314.595} C_VEL
LIN {X 0,Y 587.552,Z 305.846,A -85,B 0,C 180,E1 -1315.141,E2 -1315.141} C_VEL
LIN {X 0,Y 587.63,Z 294.594,A -85,B 0,C 180,E1 -1315.612,E2 -1315.612} C_VEL
LIN {X 0,Y 587.696,Z 282.085,A -85,B 0,C 180,E1 -1315.997,E2 -1315.997} C_VEL
LIN {X 0,Y 587.709,Z 268.631,A -85,B 0,C 180,E1 -1316.256,E2 -1316.256} C_VEL
LIN {X 0,Y 587.814,Z 169.274,A -85,B 0,C 180,E1 -1317.476,E2 -1317.476} C_VEL
LIN {X 0,Y 587.344,Z 166.061,A -85,B 0,C 180,E1 -1317.548,E2 -1317.548} C_VEL
LIN {X 0,Y 587.423,Z 149.024,A -85,B 0,C 180,E1 -1320.428,E2 -1320.428} C_VEL
LIN {X 0,Y 587.521,Z 134.225,A -85,B 0,C 180,E1 -1322.964,E2 -1322.964} C_VEL
LIN {X 0,Y 587.3,Z 130.327,A -85,B 0,C 180,E1 -1323.672,E2 -1323.672} C_VEL
LIN {X 0,Y 587.276,Z 130.328,A -85,B 0,C 180,E1 -1325.991,E2 -1325.991} C_VEL
LIN {X 0,Y 587.308,Z 130.326,A -85,B 0,C 180,E1 -1328.968,E2 -1328.968} C_VEL
LIN {X 0,Y 587.315,Z 130.322,A -85,B 0,C 180,E1 -1331.15,E2 -1331.15} C_VEL
LIN {X 0,Y 587.28,Z 130.329,A -85,B 0,C 180,E1 -1334.024,E2 -1334.024} C_VEL
LIN {X 0,Y 587.328,Z 130.325,A -85,B 0,C 180,E1 -1336.154,E2 -1336.154} C_VEL
LIN {X 0,Y 587.294,Z 130.325,A -85,B 0,C 180,E1 -1338.962,E2 -1338.962} C_VEL
LIN {X 0,Y 587.322,Z 130.322,A -85,B 0,C 180,E1 -1341.744,E2 -1341.744} C_VEL
LIN {X 0,Y 587.329,Z 130.324,A -85,B 0,C 180,E1 -1344.507,E2 -1344.507} C_VEL
LIN {X 0,Y 587.328,Z 130.319,A -85,B 0,C 180,E1 -1347.257,E2 -1347.257} C_VEL
LIN {X 0,Y 587.377,Z 130.322,A -85,B 0,C 180,E1 -1350,E2 -1350} C_VEL
LIN {X 0,Y 587.33,Z 130.32,A -85,B 0,C 180,E1 -1352.744,E2 -1352.744} C_VEL
LIN {X 0,Y 587.325,Z 130.322,A -85,B 0,C 180,E1 -1355.493,E2 -1355.493} C_VEL
LIN {X 0,Y 587.323,Z 130.324,A -85,B 0,C 180,E1 -1358.256,E2 -1358.256} C_VEL
LIN {X 0,Y 587.293,Z 130.324,A -85,B 0,C 180,E1 -1361.107,E2 -1361.107} C_VEL
LIN {X 0,Y 587.33,Z 130.328,A -85,B 0,C 180,E1 -1363.846,E2 -1363.846} C_VEL
LIN {X 0,Y 587.288,Z 130.324,A -85,B 0,C 180,E1 -1366.795,E2 -1366.795} C_VEL
LIN {X 0,Y 587.291,Z 130.333,A -85,B 0,C 180,E1 -1369.577,E2 -1369.577} C_VEL
LIN {X 0,Y 587.288,Z 130.331,A -85,B 0,C 180,E1 -1371.775,E2 -1371.775} C_VEL
LIN {X 0,Y 587.295,Z 130.324,A -85,B 0,C 180,E1 -1374.761,E2 -1374.761} C_VEL
LIN {X 0,Y 587.29,Z 130.33,A -85,B 0,C 180,E1 -1377.682,E2 -1377.682} C_VEL
LIN {X 0,Y 587.282,Z 130.325,A -85,B 0,C 180,E1 -1380.501,E2 -1380.501} C_VEL
LIN {X 0,Y 587.324,Z 130.326,A -85,B 0,C 180,E1 -1383.11,E2 -1383.11} C_VEL
LIN {X 0,Y 587.266,Z 130.328,A -85,B 0,C 180,E1 -1385.901,E2 -1385.901} C_VEL
LIN {X 0,Y 587.295,Z 130.324,A -85,B 0,C 180,E1 -1388.482,E2 -1388.482} C_VEL
LIN {X 0,Y 587.302,Z 130.333,A -85,B 0,C 180,E1 -1391.159,E2 -1391.159} C_VEL
LIN {X 0,Y 587.296,Z 130.323,A -85,B 0,C 180,E1 -1394.111,E2 -1394.111} C_VEL
LIN {X 0,Y 587.28,Z 130.335,A -85,B 0,C 180,E1 -1396.991,E2 -1396.991} C_VEL
LIN {X 0,Y 587.284,Z 130.325,A -85,B 0,C 180,E1 -1399.744,E2 -1399.744} C_VEL
LIN {X 0,Y 587.323,Z 130.322,A -85,B 0,C 180,E1 -1402.391,E2 -1402.391} C_VEL
LIN {X 0,Y 587.307,Z 130.322,A -85,B 0,C 180,E1 -1405.777,E2 -1405.777} C_VEL
LIN {X 0,Y 587.307,Z 130.324,A -85,B 0,C 180,E1 -1408.229,E2 -1408.229} C_VEL
LIN {X 0,Y 587.291,Z 130.331,A -85,B 0,C 180,E1 -1410.876,E2 -1410.876} C_VEL
LIN {X 0,Y 587.295,Z 130.323,A -85,B 0,C 180,E1 -1413.83,E2 -1413.83} C_VEL
LIN {X 0,Y 587.279,Z 130.333,A -85,B 0,C 180,E1 -1416.74,E2 -1416.74} C_VEL
LIN {X 0,Y 587.291,Z 130.324,A -85,B 0,C 180,E1 -1419.694,E2 -1419.694} C_VEL
LIN {X 0,Y 587.264,Z 130.329,A -85,B 0,C 180,E1 -1421.872,E2 -1421.872} C_VEL
LIN {X 0,Y 587.289,Z 130.329,A -85,B 0,C 180,E1 -1424.736,E2 -1424.736} C_VEL
LIN {X 0,Y 587.262,Z 130.33,A -85,B 0,C 180,E1 -1426.857,E2 -1426.857} C_VEL
LIN {X 0,Y 587.309,Z 130.323,A -85,B 0,C 180,E1 -1429.66,E2 -1429.66} C_VEL
LIN {X 0,Y 587.304,Z 130.329,A -85,B 0,C 180,E1 -1432.436,E2 -1432.436} C_VEL
LIN {X 0,Y 587.315,Z 130.321,A -85,B 0,C 180,E1 -1435.195,E2 -1435.195} C_VEL
LIN {X 0,Y 587.366,Z 130.322,A -85,B 0,C 180,E1 -1437.943,E2 -1437.943} C_VEL
LIN {X 0,Y 587.374,Z 130.323,A -85,B 0,C 180,E1 -1440,E2 -1440} C_VEL
LIN {X 0,Y 587.327,Z 130.32,A -85,B 0,C 180,E1 -1442.744,E2 -1442.744} C_VEL
LIN {X 0,Y 587.323,Z 130.323,A -85,B 0,C 180,E1 -1445.494,E2 -1445.494} C_VEL
LIN {X 0,Y 587.32,Z 130.324,A -85,B 0,C 180,E1 -1448.256,E2 -1448.256} C_VEL
LIN {X 0,Y 587.309,Z 130.322,A -85,B 0,C 180,E1 -1451.117,E2 -1451.117} C_VEL
LIN {X 0,Y 587.311,Z 130.324,A -85,B 0,C 180,E1 -1454.242,E2 -1454.242} C_VEL
LIN {X 0,Y 587.286,Z 130.324,A -85,B 0,C 180,E1 -1456.796,E2 -1456.796} C_VEL
LIN {X 0,Y 587.288,Z 130.334,A -85,B 0,C 180,E1 -1459.577,E2 -1459.577} C_VEL
LIN {X 0,Y 587.286,Z 130.331,A -85,B 0,C 180,E1 -1461.776,E2 -1461.776} C_VEL
LIN {X 0,Y 587.291,Z 130.324,A -85,B 0,C 180,E1 -1464.762,E2 -1464.762} C_VEL
LIN {X 0,Y 587.29,Z 130.33,A -85,B 0,C 180,E1 -1467.683,E2 -1467.683} C_VEL
LIN {X 0,Y 587.282,Z 130.325,A -85,B 0,C 180,E1 -1470.502,E2 -1470.502} C_VEL
LIN {X 0,Y 587.325,Z 130.326,A -85,B 0,C 180,E1 -1473.111,E2 -1473.111} C_VEL
LIN {X 0,Y 587.257,Z 130.329,A -85,B 0,C 180,E1 -1475.903,E2 -1475.903} C_VEL
LIN {X 0,Y 587.295,Z 130.324,A -85,B 0,C 180,E1 -1478.482,E2 -1478.482} C_VEL
LIN {X 0,Y 587.302,Z 130.332,A -85,B 0,C 180,E1 -1481.16,E2 -1481.16} C_VEL
LIN {X 0,Y 587.299,Z 130.323,A -85,B 0,C 180,E1 -1484.111,E2 -1484.111} C_VEL
LIN {X 0,Y 587.28,Z 130.335,A -85,B 0,C 180,E1 -1486.991,E2 -1486.991} C_VEL
LIN {X 0,Y 587.288,Z 130.324,A -85,B 0,C 180,E1 -1489.744,E2 -1489.744} C_VEL
LIN {X 0,Y 587.326,Z 130.322,A -85,B 0,C 180,E1 -1492.391,E2 -1492.391} C_VEL
LIN {X 0,Y 587.31,Z 130.321,A -85,B 0,C 180,E1 -1495.777,E2 -1495.777} C_VEL
LIN {X 0,Y 587.297,Z 130.325,A -85,B 0,C 180,E1 -1498.229,E2 -1498.229} C_VEL
LIN {X 0,Y 587.296,Z 130.33,A -85,B 0,C 180,E1 -1500.877,E2 -1500.877} C_VEL
LIN {X 0,Y 587.294,Z 130.324,A -85,B 0,C 180,E1 -1503.833,E2 -1503.833} C_VEL
LIN {X 0,Y 587.283,Z 130.335,A -85,B 0,C 180,E1 -1506.74,E2 -1506.74} C_VEL
LIN {X 0,Y 587.285,Z 130.437,A -85,B 0,C 180,E1 -1507.268,E2 -1507.268} C_VEL
LIN {X 0,Y 587.771,Z 135.745,A -85,B 0,C 180,E1 -1508.059,E2 -1508.059} C_VEL
LIN {X 0,Y 587.671,Z 155.132,A -85,B 0,C 180,E1 -1510.869,E2 -1510.869} C_VEL
LIN {X 0,Y 587.538,Z 176.061,A -85,B 0,C 180,E1 -1513.853,E2 -1513.853} C_VEL
LIN {X 0,Y 587.425,Z 195.149,A -85,B 0,C 180,E1 -1516.509,E2 -1516.509} C_VEL
LIN {X 0,Y 587.843,Z 200.515,A -85,B 0,C 180,E1 -1516.584,E2 -1516.584} C_VEL
LIN {X 0,Y 587.729,Z 302.95,A -85,B 0,C 180,E1 -1517.855,E2 -1517.855} C_VEL
LIN {X 0,Y 587.668,Z 316.222,A -85,B 0,C 180,E1 -1518.16,E2 -1518.16} C_VEL
LIN {X 0,Y 587.6,Z 328.774,A -85,B 0,C 180,E1 -1518.59,E2 -1518.59} C_VEL
LIN {X 0,Y 587.536,Z 340.63,A -85,B 0,C 180,E1 -1519.141,E2 -1519.141} C_VEL
LIN {X 0,Y 587.464,Z 352.204,A -85,B 0,C 180,E1 -1519.836,E2 -1519.836} C_VEL
LIN {X 0,Y 587.366,Z 362.599,A -85,B 0,C 180,E1 -1520.617,E2 -1520.617} C_VEL
LIN {X 0,Y 587.322,Z 371.113,A -85,B 0,C 180,E1 -1521.398,E2 -1521.398} C_VEL
LIN {X 0,Y 587.274,Z 378.961,A -85,B 0,C 180,E1 -1522.263,E2 -1522.263} C_VEL
LIN {X 0,Y 587.23,Z 385.469,A -85,B 0,C 180,E1 -1523.126,E2 -1523.126} C_VEL
LIN {X 0,Y 587.237,Z 391.866,A -85,B 0,C 180,E1 -1524.161,E2 -1524.161} C_VEL
LIN {X 0,Y 587.147,Z 396.95,A -85,B 0,C 180,E1 -1525.194,E2 -1525.194} C_VEL
LIN {X 0,Y 587.213,Z 400.895,A -85,B 0,C 180,E1 -1526.226,E2 -1526.226} C_VEL
LIN {X 0,Y 587.132,Z 403.808,A -85,B 0,C 180,E1 -1527.256,E2 -1527.256} C_VEL
LIN {X 0,Y 587.141,Z 405.199,A -85,B 0,C 180,E1 -1527.942,E2 -1527.942} C_VEL
LIN {X 0,Y 587.14,Z 406.784,A -85,B 0,C 180,E1 -1529.314,E2 -1529.314} C_VEL
LIN {X 0,Y 587.137,Z 407,A -85,B 0,C 180,E1 -1530,E2 -1530} C_VEL
LIN {X 0,Y 587.147,Z 406.186,A -85,B 0,C 180,E1 -1531.372,E2 -1531.372} C_VEL
LIN {X 0,Y 587.141,Z 405.201,A -85,B 0,C 180,E1 -1532.058,E2 -1532.058} C_VEL
LIN {X 0,Y 587.132,Z 403.81,A -85,B 0,C 180,E1 -1532.744,E2 -1532.744} C_VEL
LIN {X 0,Y 587.213,Z 400.896,A -85,B 0,C 180,E1 -1533.774,E2 -1533.774} C_VEL
LIN {X 0,Y 587.147,Z 396.95,A -85,B 0,C 180,E1 -1534.806,E2 -1534.806} C_VEL
LIN {X 0,Y 587.218,Z 390.878,A -85,B 0,C 180,E1 -1536.011,E2 -1536.011} C_VEL
LIN {X 0,Y 587.245,Z 384.239,A -85,B 0,C 180,E1 -1537.046,E2 -1537.046} C_VEL
LIN {X 0,Y 587.299,Z 375.992,A -85,B 0,C 180,E1 -1538.083,E2 -1538.083} C_VEL
LIN {X 0,Y 587.343,Z 367.541,A -85,B 0,C 180,E1 -1538.949,E2 -1538.949} C_VEL
LIN {X 0,Y 587.419,Z 357.1,A -85,B 0,C 180,E1 -1539.816,E2 -1539.816} C_VEL
LIN {X 0,Y 587.497,Z 346.76,A -85,B 0,C 180,E1 -1540.511,E2 -1540.511} C_VEL
LIN {X 0,Y 587.561,Z 334.822,A -85,B 0,C 180,E1 -1541.149,E2 -1541.149} C_VEL
LIN {X 0,Y 587.629,Z 322.607,A -85,B 0,C 180,E1 -1541.639,E2 -1541.639} C_VEL
LIN {X 0,Y 587.704,Z 309.447,A -85,B 0,C 180,E1 -1542.014,E2 -1542.014} C_VEL
LIN {X 0,Y 587.778,Z 297.106,A -85,B 0,C 180,E1 -1542.231,E2 -1542.231} C_VEL
LIN {X 0,Y 587.703,Z 196.958,A -85,B 0,C 180,E1 -1543.463,E2 -1543.463} C_VEL
LIN {X 0,Y 587.381,Z 194.795,A -85,B 0,C 180,E1 -1543.514,E2 -1543.514} C_VEL
LIN {X 0,Y 587.542,Z 174.803,A -85,B 0,C 180,E1 -1546.325,E2 -1546.325} C_VEL
LIN {X 0,Y 587.67,Z 155.133,A -85,B 0,C 180,E1 -1549.131,E2 -1549.131} C_VEL
LIN {X 0,Y 587.77,Z 135.738,A -85,B 0,C 180,E1 -1551.941,E2 -1551.941} C_VEL
LIN {X 0,Y 587.276,Z 130.376,A -85,B 0,C 180,E1 -1552.732,E2 -1552.732} C_VEL
LIN {X 0,Y 587.295,Z 130.332,A -85,B 0,C 180,E1 -1555.518,E2 -1555.518} C_VEL
LIN {X 0,Y 587.283,Z 130.329,A -85,B 0,C 180,E1 -1557.82,E2 -1557.82} C_VEL
LIN {X 0,Y 587.284,Z 130.326,A -85,B 0,C 180,E1 -1560.501,E2 -1560.501} C_VEL
LIN {X 0,Y 587.286,Z 130.333,A -85,B 0,C 180,E1 -1563.103,E2 -1563.103} C_VEL
LIN {X 0,Y 587.248,Z 130.334,A -85,B 0,C 180,E1 -1565.53,E2 -1565.53} C_VEL
LIN {X 0,Y 587.307,Z 130.323,A -85,B 0,C 180,E1 -1567.834,E2 -1567.834} C_VEL
LIN {X 0,Y 587.286,Z 130.325,A -85,B 0,C 180,E1 -1570.256,E2 -1570.256} C_VEL
LIN {X 0,Y 587.281,Z 130.334,A -85,B 0,C 180,E1 -1573.114,E2 -1573.114} C_VEL
LIN {X 0,Y 587.293,Z 130.324,A -85,B 0,C 180,E1 -1576.046,E2 -1576.046} C_VEL
LIN {X 0,Y 587.301,Z 130.332,A -85,B 0,C 180,E1 -1578.928,E2 -1578.928} C_VEL
LIN {X 0,Y 587.294,Z 130.324,A -85,B 0,C 180,E1 -1581.518,E2 -1581.518} C_VEL
LIN {X 0,Y 587.256,Z 130.329,A -85,B 0,C 180,E1 -1584.097,E2 -1584.097} C_VEL
LIN {X 0,Y 587.323,Z 130.326,A -85,B 0,C 180,E1 -1586.889,E2 -1586.889} C_VEL
LIN {X 0,Y 587.285,Z 130.324,A -85,B 0,C 180,E1 -1589.827,E2 -1589.827} C_VEL
LIN {X 0,Y 587.292,Z 130.327,A -85,B 0,C 180,E1 -1592.952,E2 -1592.952} C_VEL
LIN {X 0,Y 587.285,Z 130.325,A -85,B 0,C 180,E1 -1595.432,E2 -1595.432} C_VEL
LIN {X 0,Y 587.285,Z 130.33,A -85,B 0,C 180,E1 -1598.224,E2 -1598.224} C_VEL
LIN {X 0,Y 587.31,Z 130.321,A -85,B 0,C 180,E1 -1601.15,E2 -1601.15} C_VEL
LIN {X 0,Y 587.277,Z 130.331,A -85,B 0,C 180,E1 -1604.023,E2 -1604.023} C_VEL
LIN {X 0,Y 587.324,Z 130.328,A -85,B 0,C 180,E1 -1606.153,E2 -1606.153} C_VEL
LIN {X 0,Y 587.289,Z 130.325,A -85,B 0,C 180,E1 -1608.961,E2 -1608.961} C_VEL
LIN {X 0,Y 587.318,Z 130.324,A -85,B 0,C 180,E1 -1611.744,E2 -1611.744} C_VEL
LIN {X 0,Y 587.322,Z 130.323,A -85,B 0,C 180,E1 -1614.506,E2 -1614.506} C_VEL
LIN {X 0,Y 587.325,Z 130.32,A -85,B 0,C 180,E1 -1617.256,E2 -1617.256} C_VEL
LIN {X 0,Y 587.372,Z 130.323,A -85,B 0,C 180,E1 -1620,E2 -1620} C_VEL
LIN {X 0,Y 587.324,Z 130.32,A -85,B 0,C 180,E1 -1622.743,E2 -1622.743} C_VEL
LIN {X 0,Y 587.325,Z 130.324,A -85,B 0,C 180,E1 -1625.493,E2 -1625.493} C_VEL
LIN {X 0,Y 587.317,Z 130.324,A -85,B 0,C 180,E1 -1628.256,E2 -1628.256} C_VEL
LIN {X 0,Y 587.305,Z 130.325,A -85,B 0,C 180,E1 -1631.116,E2 -1631.116} C_VEL
LIN {X 0,Y 587.323,Z 130.328,A -85,B 0,C 180,E1 -1633.846,E2 -1633.846} C_VEL
LIN {X 0,Y 587.265,Z 130.328,A -85,B 0,C 180,E1 -1636.79,E2 -1636.79} C_VEL
LIN {X 0,Y 587.264,Z 130.328,A -85,B 0,C 180,E1 -1638.267,E2 -1638.267} C_VEL
LIN {X 0,Y 586.614,Z 130.41,A -85,B 0,C 180,E1 -1638.839,E2 -1638.839} C_VEL
LIN {X 0,Y 583.768,Z 130.769,A -85,B 0,C 180,E1 -1639.767,E2 -1639.767} C_VEL
LIN {X 0,Y 581.362,Z 131.066,A -85,B 0,C 180,E1 -1640.514,E2 -1640.514} C_VEL
LIN {X 0,Y 580.34,Z 131.195,A -85,B 0,C 180,E1 -1641.091,E2 -1641.091} C_VEL
LIN {X 0,Y 580.263,Z 131.207,A -85,B 0,C 180,E1 -1641.286,E2 -1641.286} C_VEL
LIN {X 0,Y 580.255,Z 131.279,A -85,B 0,C 180,E1 -1644.377,E2 -1644.377} C_VEL
LIN {X 0,Y 580.533,Z 136.346,A -85,B 0,C 180,E1 -1645.261,E2 -1645.261} C_VEL
LIN {X 0,Y 580.385,Z 153.224,A -85,B 0,C 180,E1 -1648.181,E2 -1648.181} C_VEL
LIN {X 0,Y 580.346,Z 166.175,A -85,B 0,C 180,E1 -1650.395,E2 -1650.395} C_VEL
LIN {X 0,Y 580.974,Z 171.872,A -85,B 0,C 180,E1 -1650.485,E2 -1650.485} C_VEL
LIN {X 0,Y 580.79,Z 273.424,A -85,B 0,C 180,E1 -1651.761,E2 -1651.761} C_VEL
LIN {X 0,Y 580.713,Z 285.59,A -85,B 0,C 180,E1 -1652.047,E2 -1652.047} C_VEL
LIN {X 0,Y 580.649,Z 297.15,A -85,B 0,C 180,E1 -1652.435,E2 -1652.435} C_VEL
LIN {X 0,Y 580.53,Z 309.815,A -85,B 0,C 180,E1 -1653.009,E2 -1653.009} C_VEL
LIN {X 0,Y 580.434,Z 321.375,A -85,B 0,C 180,E1 -1653.703,E2 -1653.703} C_VEL
LIN {X 0,Y 580.369,Z 330.954,A -85,B 0,C 180,E1 -1654.417,E2 -1654.417} C_VEL
LIN {X 0,Y 580.288,Z 339.934,A -85,B 0,C 180,E1 -1655.225,E2 -1655.225} C_VEL
LIN {X 0,Y 580.206,Z 349.106,A -85,B 0,C 180,E1 -1656.232,E2 -1656.232} C_VEL
LIN {X 0,Y 580.159,Z 356.731,A -85,B 0,C 180,E1 -1657.279,E2 -1657.279} C_VEL
LIN {X 0,Y 580.124,Z 363.13,A -85,B 0,C 180,E1 -1658.38,E2 -1658.38} C_VEL
LIN {X 0,Y 580.084,Z 366.852,A -85,B 0,C 180,E1 -1659.161,E2 -1659.161} C_VEL
LIN {X 0,Y 580.099,Z 370.941,A -85,B 0,C 180,E1 -1660.249,E2 -1660.249} C_VEL
LIN {X 0,Y 580.035,Z 373.859,A -85,B 0,C 180,E1 -1661.305,E2 -1661.305} C_VEL
LIN {X 0,Y 580.057,Z 375.781,A -85,B 0,C 180,E1 -1662.348,E2 -1662.348} C_VEL
LIN {X 0,Y 580.021,Z 376.912,A -85,B 0,C 180,E1 -1663.682,E2 -1663.682} C_VEL
LIN {X 0,Y 580.064,Z 376.811,A -85,B 0,C 180,E1 -1664.645,E2 -1664.645} C_VEL
LIN {X 0,Y 580.06,Z 375.924,A -85,B 0,C 180,E1 -1665.63,E2 -1665.63} C_VEL
LIN {X 0,Y 580.029,Z 374.181,A -85,B 0,C 180,E1 -1666.635,E2 -1666.635} C_VEL
LIN {X 0,Y 580.08,Z 371.522,A -85,B 0,C 180,E1 -1667.65,E2 -1667.65} C_VEL
LIN {X 0,Y 580.076,Z 367.82,A -85,B 0,C 180,E1 -1668.691,E2 -1668.691} C_VEL
LIN {X 0,Y 580.126,Z 362.938,A -85,B 0,C 180,E1 -1669.748,E2 -1669.748} C_VEL
LIN {X 0,Y 580.182,Z 355.774,A -85,B 0,C 180,E1 -1670.958,E2 -1670.958} C_VEL
LIN {X 0,Y 580.203,Z 348.432,A -85,B 0,C 180,E1 -1671.938,E2 -1671.938} C_VEL
LIN {X 0,Y 580.301,Z 341.275,A -85,B 0,C 180,E1 -1672.733,E2 -1672.733} C_VEL
LIN {X 0,Y 580.376,Z 332.933,A -85,B 0,C 180,E1 -1673.509,E2 -1673.509} C_VEL
LIN {X 0,Y 580.402,Z 323.746,A -85,B 0,C 180,E1 -1674.222,E2 -1674.222} C_VEL
LIN {X 0,Y 580.474,Z 314.972,A -85,B 0,C 180,E1 -1674.788,E2 -1674.788} C_VEL
LIN {X 0,Y 580.591,Z 304.783,A -85,B 0,C 180,E1 -1675.325,E2 -1675.325} C_VEL
LIN {X 0,Y 580.67,Z 293.197,A -85,B 0,C 180,E1 -1675.803,E2 -1675.803} C_VEL
LIN {X 0,Y 580.746,Z 279.451,A -85,B 0,C 180,E1 -1676.206,E2 -1676.206} C_VEL
LIN {X 0,Y 580.808,Z 266.41,A -85,B 0,C 180,E1 -1676.434,E2 -1676.434} C_VEL
LIN {X 0,Y 580.895,Z 169.859,A -85,B 0,C 180,E1 -1677.632,E2 -1677.632} C_VEL
LIN {X 0,Y 580.314,Z 166.156,A -85,B 0,C 180,E1 -1677.699,E2 -1677.699} C_VEL
LIN {X 0,Y 580.455,Z 148.839,A -85,B 0,C 180,E1 -1680.663,E2 -1680.663} C_VEL
LIN {X 0,Y 580.553,Z 133.141,A -85,B 0,C 180,E1 -1683.391,E2 -1683.391} C_VEL
LIN {X 0,Y 580.267,Z 131.204,A -85,B 0,C 180,E1 -1683.746,E2 -1683.746} C_VEL
LIN {X 0,Y 580.236,Z 131.211,A -85,B 0,C 180,E1 -1686.441,E2 -1686.441} C_VEL
LIN {X 0,Y 580.243,Z 131.202,A -85,B 0,C 180,E1 -1689.436,E2 -1689.436} C_VEL
LIN {X 0,Y 580.228,Z 131.204,A -85,B 0,C 180,E1 -1691.644,E2 -1691.644} C_VEL
LIN {X 0,Y 580.259,Z 131.208,A -85,B 0,C 180,E1 -1694.547,E2 -1694.547} C_VEL
LIN {X 0,Y 580.227,Z 131.209,A -85,B 0,C 180,E1 -1696.695,E2 -1696.695} C_VEL
LIN {X 0,Y 580.264,Z 131.202,A -85,B 0,C 180,E1 -1698.826,E2 -1698.826} C_VEL
LIN {X 0,Y 580.289,Z 131.197,A -85,B 0,C 180,E1 -1701.644,E2 -1701.644} C_VEL
LIN {X 0,Y 580.297,Z 131.201,A -85,B 0,C 180,E1 -1704.44,E2 -1704.44} C_VEL
LIN {X 0,Y 580.336,Z 131.196,A -85,B 0,C 180,E1 -1707.918,E2 -1707.918} C_VEL
LIN {X 0,Y 580.345,Z 131.198,A -85,B 0,C 180,E1 -1710,E2 -1710} C_VEL
LIN {X 0,Y 580.298,Z 131.195,A -85,B 0,C 180,E1 -1712.777,E2 -1712.777} C_VEL
LIN {X 0,Y 580.294,Z 131.199,A -85,B 0,C 180,E1 -1715.56,E2 -1715.56} C_VEL
LIN {X 0,Y 580.289,Z 131.199,A -85,B 0,C 180,E1 -1718.357,E2 -1718.357} C_VEL
LIN {X 0,Y 580.264,Z 131.2,A -85,B 0,C 180,E1 -1721.174,E2 -1721.174} C_VEL
LIN {X 0,Y 580.289,Z 131.202,A -85,B 0,C 180,E1 -1724.018,E2 -1724.018} C_VEL
LIN {X 0,Y 580.246,Z 131.202,A -85,B 0,C 180,E1 -1726.899,E2 -1726.899} C_VEL
LIN {X 0,Y 580.264,Z 131.206,A -85,B 0,C 180,E1 -1729.824,E2 -1729.824} C_VEL
LIN {X 0,Y 580.223,Z 131.207,A -85,B 0,C 180,E1 -1732.054,E2 -1732.054} C_VEL
LIN {X 0,Y 580.274,Z 131.201,A -85,B 0,C 180,E1 -1735.081,E2 -1735.081} C_VEL
LIN {X 0,Y 580.234,Z 131.207,A -85,B 0,C 180,E1 -1737.847,E2 -1737.847} C_VEL
LIN {X 0,Y 580.239,Z 131.203,A -85,B 0,C 180,E1 -1740.687,E2 -1740.687} C_VEL
LIN {X 0,Y 580.27,Z 131.208,A -85,B 0,C 180,E1 -1743.312,E2 -1743.312} C_VEL
LIN {X 0,Y 580.216,Z 131.208,A -85,B 0,C 180,E1 -1745.753,E2 -1745.753} C_VEL
LIN {X 0,Y 580.267,Z 131.199,A -85,B 0,C 180,E1 -1748.147,E2 -1748.147} C_VEL
LIN {X 0,Y 580.249,Z 131.206,A -85,B 0,C 180,E1 -1750.847,E2 -1750.847} C_VEL
LIN {X 0,Y 580.229,Z 131.205,A -85,B 0,C 180,E1 -1753.662,E2 -1753.662} C_VEL
LIN {X 0,Y 580.228,Z 131.204,A -85,B 0,C 180,E1 -1756.338,E2 -1756.338} C_VEL
LIN {X 0,Y 580.268,Z 131.206,A -85,B 0,C 180,E1 -1759.154,E2 -1759.154} C_VEL
LIN {X 0,Y 580.268,Z 131.198,A -85,B 0,C 180,E1 -1761.929,E2 -1761.929} C_VEL
LIN {X 0,Y 580.209,Z 131.21,A -85,B 0,C 180,E1 -1764.45,E2 -1764.45} C_VEL
LIN {X 0,Y 580.273,Z 131.205,A -85,B 0,C 180,E1 -1766.974,E2 -1766.974} C_VEL
LIN {X 0,Y 580.259,Z 131.201,A -85,B 0,C 180,E1 -1769.423,E2 -1769.423} C_VEL
LIN {X 0,Y 580.231,Z 131.205,A -85,B 0,C 180,E1 -1772.153,E2 -1772.153} C_VEL
LIN {X 0,Y 580.267,Z 131.204,A -85,B 0,C 180,E1 -1774.919,E2 -1774.919} C_VEL
LIN {X 0,Y 580.222,Z 131.206,A -85,B 0,C 180,E1 -1777.946,E2 -1777.946} C_VEL
LIN {X 0,Y 580.267,Z 131.202,A -85,B 0,C 180,E1 -1780.913,E2 -1780.913} C_VEL
LIN {X 0,Y 580.228,Z 131.205,A -85,B 0,C 180,E1 -1783.824,E2 -1783.824} C_VEL
LIN {X 0,Y 580.284,Z 131.2,A -85,B 0,C 180,E1 -1785.982,E2 -1785.982} C_VEL
LIN {X 0,Y 580.26,Z 131.202,A -85,B 0,C 180,E1 -1788.826,E2 -1788.826} C_VEL
LIN {X 0,Y 580.285,Z 131.198,A -85,B 0,C 180,E1 -1791.644,E2 -1791.644} C_VEL
LIN {X 0,Y 580.294,Z 131.201,A -85,B 0,C 180,E1 -1794.44,E2 -1794.44} C_VEL
LIN {X 0,Y 580.334,Z 131.197,A -85,B 0,C 180,E1 -1797.918,E2 -1797.918} C_VEL
LIN {X 0,Y 580.342,Z 131.199,A -85,B 0,C 180,E1 -1800,E2 -1800} C_VEL
LIN {X 0,Y 580.295,Z 131.196,A -85,B 0,C 180,E1 -1802.777,E2 -1802.777} C_VEL
LIN {X 0,Y 580.292,Z 131.2,A -85,B 0,C 180,E1 -1805.56,E2 -1805.56} C_VEL
LIN {X 0,Y 580.286,Z 131.199,A -85,B 0,C 180,E1 -1808.357,E2 -1808.357} C_VEL
LIN {X 0,Y 580.261,Z 131.201,A -85,B 0,C 180,E1 -1811.174,E2 -1811.174} C_VEL
LIN {X 0,Y 580.285,Z 131.202,A -85,B 0,C 180,E1 -1814.018,E2 -1814.018} C_VEL
LIN {X 0,Y 580.244,Z 131.202,A -85,B 0,C 180,E1 -1816.9,E2 -1816.9} C_VEL
LIN {X 0,Y 580.262,Z 131.206,A -85,B 0,C 180,E1 -1819.824,E2 -1819.824} C_VEL
LIN {X 0,Y 580.221,Z 131.207,A -85,B 0,C 180,E1 -1822.055,E2 -1822.055} C_VEL
LIN {X 0,Y 580.27,Z 131.202,A -85,B 0,C 180,E1 -1825.082,E2 -1825.082} C_VEL
LIN {X 0,Y 580.233,Z 131.207,A -85,B 0,C 180,E1 -1827.848,E2 -1827.848} C_VEL
LIN {X 0,Y 580.235,Z 131.204,A -85,B 0,C 180,E1 -1830.687,E2 -1830.687} C_VEL
LIN {X 0,Y 580.271,Z 131.209,A -85,B 0,C 180,E1 -1833.312,E2 -1833.312} C_VEL
LIN {X 0,Y 580.208,Z 131.209,A -85,B 0,C 180,E1 -1835.752,E2 -1835.752} C_VEL
LIN {X 0,Y 580.268,Z 131.199,A -85,B 0,C 180,E1 -1838.148,E2 -1838.148} C_VEL
LIN {X 0,Y 580.249,Z 131.206,A -85,B 0,C 180,E1 -1840.848,E2 -1840.848} C_VEL
LIN {X 0,Y 580.231,Z 131.205,A -85,B 0,C 180,E1 -1843.663,E2 -1843.663} C_VEL
LIN {X 0,Y 580.231,Z 131.204,A -85,B 0,C 180,E1 -1846.338,E2 -1846.338} C_VEL
LIN {X 0,Y 580.25,Z 131.208,A -85,B 0,C 180,E1 -1849.153,E2 -1849.153} C_VEL
LIN {X 0,Y 580.272,Z 131.198,A -85,B 0,C 180,E1 -1851.93,E2 -1851.93} C_VEL
LIN {X 0,Y 580.204,Z 131.21,A -85,B 0,C 180,E1 -1854.45,E2 -1854.45} C_VEL
LIN {X 0,Y 580.24,Z 131.209,A -85,B 0,C 180,E1 -1856.972,E2 -1856.972} C_VEL
LIN {X 0,Y 580.249,Z 131.202,A -85,B 0,C 180,E1 -1859.423,E2 -1859.423} C_VEL
LIN {X 0,Y 580.237,Z 131.205,A -85,B 0,C 180,E1 -1862.153,E2 -1862.153} C_VEL
LIN {X 0,Y 580.238,Z 131.208,A -85,B 0,C 180,E1 -1864.917,E2 -1864.917} C_VEL
LIN {X 0,Y 580.267,Z 131.398,A -85,B 0,C 180,E1 -1867.142,E2 -1867.142} C_VEL
LIN {X 0,Y 580.833,Z 135.602,A -85,B 0,C 180,E1 -1867.783,E2 -1867.783} C_VEL
LIN {X 0,Y 580.709,Z 154.386,A -85,B 0,C 180,E1 -1870.521,E2 -1870.521} C_VEL
LIN {X 0,Y 580.537,Z 173.542,A -85,B 0,C 180,E1 -1873.291,E2 -1873.291} C_VEL
LIN {X 0,Y 580.401,Z 194.635,A -85,B 0,C 180,E1 -1876.298,E2 -1876.298} C_VEL
LIN {X 0,Y 580.399,Z 195.149,A -85,B 0,C 180,E1 -1876.342,E2 -1876.342} C_VEL
LIN {X 0,Y 580.95,Z 200.515,A -85,B 0,C 180,E1 -1876.422,E2 -1876.422} C_VEL
LIN {X 0,Y 580.811,Z 302.95,A -85,B 0,C 180,E1 -1877.708,E2 -1877.708} C_VEL
LIN {X 0,Y 580.727,Z 316.221,A -85,B 0,C 180,E1 -1878.017,E2 -1878.017} C_VEL
LIN {X 0,Y 580.647,Z 328.376,A -85,B 0,C 180,E1 -1878.436,E2 -1878.436} C_VEL
LIN {X 0,Y 580.542,Z 340.628,A -85,B 0,C 180,E1 -1879.008,E2 -1879.008} C_VEL
LIN {X 0,Y 580.441,Z 352.201,A -85,B 0,C 180,E1 -1879.712,E2 -1879.712} C_VEL
LIN {X 0,Y 580.345,Z 362.601,A -85,B 0,C 180,E1 -1880.503,E2 -1880.503} C_VEL
LIN {X 0,Y 580.271,Z 371.113,A -85,B 0,C 180,E1 -1881.292,E2 -1881.292} C_VEL
LIN {X 0,Y 580.222,Z 378.961,A -85,B 0,C 180,E1 -1882.168,E2 -1882.168} C_VEL
LIN {X 0,Y 580.154,Z 386.651,A -85,B 0,C 180,E1 -1883.222,E2 -1883.222} C_VEL
LIN {X 0,Y 580.139,Z 393.68,A -85,B 0,C 180,E1 -1884.438,E2 -1884.438} C_VEL
LIN {X 0,Y 580.108,Z 398.372,A -85,B 0,C 180,E1 -1885.483,E2 -1885.483} C_VEL
LIN {X 0,Y 580.123,Z 401.957,A -85,B 0,C 180,E1 -1886.527,E2 -1886.527} C_VEL
LIN {X 0,Y 580.043,Z 403.808,A -85,B 0,C 180,E1 -1887.222,E2 -1887.222} C_VEL
LIN {X 0,Y 580.04,Z 405.198,A -85,B 0,C 180,E1 -1887.917,E2 -1887.917} C_VEL
LIN {X 0,Y 580.04,Z 406.785,A -85,B 0,C 180,E1 -1889.306,E2 -1889.306} C_VEL
LIN {X 0,Y 580.037,Z 407,A -85,B 0,C 180,E1 -1890,E2 -1890} C_VEL
LIN {X 0,Y 580.047,Z 406.186,A -85,B 0,C 180,E1 -1891.388,E2 -1891.388} C_VEL
LIN {X 0,Y 580.04,Z 405.2,A -85,B 0,C 180,E1 -1892.083,E2 -1892.083} C_VEL
LIN {X 0,Y 580.043,Z 403.81,A -85,B 0,C 180,E1 -1892.778,E2 -1892.778} C_VEL
LIN {X 0,Y 580.11,Z 400.896,A -85,B 0,C 180,E1 -1893.82,E2 -1893.82} C_VEL
LIN {X 0,Y 580.053,Z 396.95,A -85,B 0,C 180,E1 -1894.865,E2 -1894.865} C_VEL
LIN {X 0,Y 580.139,Z 390.878,A -85,B 0,C 180,E1 -1896.085,E2 -1896.085} C_VEL
LIN {X 0,Y 580.184,Z 384.239,A -85,B 0,C 180,E1 -1897.132,E2 -1897.132} C_VEL
LIN {X 0,Y 580.25,Z 375.993,A -85,B 0,C 180,E1 -1898.182,E2 -1898.182} C_VEL
LIN {X 0,Y 580.308,Z 367.541,A -85,B 0,C 180,E1 -1899.058,E2 -1899.058} C_VEL
LIN {X 0,Y 580.422,Z 357.101,A -85,B 0,C 180,E1 -1899.936,E2 -1899.936} C_VEL
LIN {X 0,Y 580.506,Z 346.758,A -85,B 0,C 180,E1 -1900.639,E2 -1900.639} C_VEL
LIN {X 0,Y 580.596,Z 335.252,A -85,B 0,C 180,E1 -1901.264,E2 -1901.264} C_VEL
LIN {X 0,Y 580.682,Z 322.48,A -85,B 0,C 180,E1 -1901.785,E2 -1901.785} C_VEL
LIN {X 0,Y 580.755,Z 309.445,A -85,B 0,C 180,E1 -1902.16,E2 -1902.16} C_VEL
LIN {X 0,Y 580.853,Z 297.106,A -85,B 0,C 180,E1 -1902.379,E2 -1902.379} C_VEL
LIN {X 0,Y 580.787,Z 197.628,A -85,B 0,C 180,E1 -1903.618,E2 -1903.618} C_VEL
LIN {X 0,Y 580.387,Z 194.795,A -85,B 0,C 180,E1 -1903.68,E2 -1903.68} C_VEL
LIN {X 0,Y 580.537,Z 174.803,A -85,B 0,C 180,E1 -1906.528,E2 -1906.528} C_VEL
LIN {X 0,Y 580.701,Z 155.857,A -85,B 0,C 180,E1 -1909.264,E2 -1909.264} C_VEL
LIN {X 0,Y 580.848,Z 138.052,A -85,B 0,C 180,E1 -1911.842,E2 -1911.842} C_VEL
LIN {X 0,Y 580.528,Z 132.903,A -85,B 0,C 180,E1 -1912.604,E2 -1912.604} C_VEL
LIN {X 0,Y 580.227,Z 131.211,A -85,B 0,C 180,E1 -1912.887,E2 -1912.887} C_VEL
LIN {X 0,Y 580.237,Z 131.209,A -85,B 0,C 180,E1 -1915.082,E2 -1915.082} C_VEL
LIN {X 0,Y 580.236,Z 131.206,A -85,B 0,C 180,E1 -1917.846,E2 -1917.846} C_VEL
LIN {X 0,Y 580.238,Z 131.206,A -85,B 0,C 180,E1 -1920.686,E2 -1920.686} C_VEL
LIN {X 0,Y 580.267,Z 131.208,A -85,B 0,C 180,E1 -1923.31,E2 -1923.31} C_VEL
LIN {X 0,Y 580.202,Z 131.209,A -85,B 0,C 180,E1 -1925.75,E2 -1925.75} C_VEL
LIN {X 0,Y 580.269,Z 131.199,A -85,B 0,C 180,E1 -1928.147,E2 -1928.147} C_VEL
LIN {X 0,Y 580.249,Z 131.208,A -85,B 0,C 180,E1 -1930.847,E2 -1930.847} C_VEL
LIN {X 0,Y 580.23,Z 131.205,A -85,B 0,C 180,E1 -1933.662,E2 -1933.662} C_VEL
LIN {X 0,Y 580.23,Z 131.206,A -85,B 0,C 180,E1 -1936.337,E2 -1936.337} C_VEL
LIN {X 0,Y 580.248,Z 131.206,A -85,B 0,C 180,E1 -1939.152,E2 -1939.152} C_VEL
LIN {X 0,Y 580.269,Z 131.199,A -85,B 0,C 180,E1 -1941.928,E2 -1941.928} C_VEL
LIN {X 0,Y 580.208,Z 131.211,A -85,B 0,C 180,E1 -1944.449,E2 -1944.449} C_VEL
LIN {X 0,Y 580.274,Z 131.203,A -85,B 0,C 180,E1 -1946.974,E2 -1946.974} C_VEL
LIN {X 0,Y 580.244,Z 131.202,A -85,B 0,C 180,E1 -1949.422,E2 -1949.422} C_VEL
LIN {X 0,Y 580.231,Z 131.207,A -85,B 0,C 180,E1 -1952.152,E2 -1952.152} C_VEL
LIN {X 0,Y 580.271,Z 131.202,A -85,B 0,C 180,E1 -1954.918,E2 -1954.918} C_VEL
LIN {X 0,Y 580.22,Z 131.206,A -85,B 0,C 180,E1 -1957.945,E2 -1957.945} C_VEL
LIN {X 0,Y 580.266,Z 131.2,A -85,B 0,C 180,E1 -1960.912,E2 -1960.912} C_VEL
LIN {X 0,Y 580.227,Z 131.207,A -85,B 0,C 180,E1 -1963.824,E2 -1963.824} C_VEL
LIN {X 0,Y 580.283,Z 131.202,A -85,B 0,C 180,E1 -1965.982,E2 -1965.982} C_VEL
LIN {X 0,Y 580.259,Z 131.201,A -85,B 0,C 180,E1 -1968.826,E2 -1968.826} C_VEL
LIN {X 0,Y 580.284,Z 131.199,A -85,B 0,C 180,E1 -1971.643,E2 -1971.643} C_VEL
LIN {X 0,Y 580.291,Z 131.199,A -85,B 0,C 180,E1 -1974.44,E2 -1974.44} C_VEL
LIN {X 0,Y 580.334,Z 131.2,A -85,B 0,C 180,E1 -1977.918,E2 -1977.918} C_VEL
LIN {X 0,Y 580.34,Z 131.199,A -85,B 0,C 180,E1 -1980,E2 -1980} C_VEL
LIN {X 0,Y 580.292,Z 131.196,A -85,B 0,C 180,E1 -1982.776,E2 -1982.776} C_VEL
LIN {X 0,Y 580.293,Z 131.201,A -85,B 0,C 180,E1 -1985.56,E2 -1985.56} C_VEL
LIN {X 0,Y 580.284,Z 131.199,A -85,B 0,C 180,E1 -1988.356,E2 -1988.356} C_VEL
LIN {X 0,Y 580.257,Z 131.203,A -85,B 0,C 180,E1 -1991.174,E2 -1991.174} C_VEL
LIN {X 0,Y 580.282,Z 131.202,A -85,B 0,C 180,E1 -1994.018,E2 -1994.018} C_VEL
LIN {X 0,Y 580.214,Z 131.207,A -85,B 0,C 180,E1 -1996.9,E2 -1996.9} C_VEL
LIN {X 0,Y 580.26,Z 131.206,A -85,B 0,C 180,E1 -1999.824,E2 -1999.824} C_VEL
LIN {X 0,Y 580.263,Z 131.207,A -85,B 0,C 180,E1 -2001.286,E2 -2001.286} C_VEL
LIN {X 0,Y 579.598,Z 131.295,A -85,B 0,C 180,E1 -2001.673,E2 -2001.673} C_VEL
LIN {X 0,Y 576.757,Z 131.65,A -85,B 0,C 180,E1 -2002.277,E2 -2002.277} C_VEL
LIN {X 0,Y 573.886,Z 132.003,A -85,B 0,C 180,E1 -2002.886,E2 -2002.886} C_VEL
LIN {X 0,Y 573.192,Z 132.086,A -85,B 0,C 180,E1 -2003.279,E2 -2003.279} C_VEL
LIN {X 0,Y 573.24,Z 132.212,A -85,B 0,C 180,E1 -2004.346,E2 -2004.346} C_VEL
LIN {X 0,Y 573.51,Z 139.435,A -85,B 0,C 180,E1 -2005.592,E2 -2005.592} C_VEL
LIN {X 0,Y 573.35,Z 156.54,A -85,B 0,C 180,E1 -2008.558,E2 -2008.558} C_VEL
LIN {X 0,Y 573.331,Z 166.154,A -85,B 0,C 180,E1 -2010.222,E2 -2010.222} C_VEL
LIN {X 0,Y 574.086,Z 172.75,A -85,B 0,C 180,E1 -2010.33,E2 -2010.33} C_VEL
LIN {X 0,Y 573.877,Z 273.144,A -85,B 0,C 180,E1 -2011.606,E2 -2011.606} C_VEL
LIN {X 0,Y 573.76,Z 285.15,A -85,B 0,C 180,E1 -2011.888,E2 -2011.888} C_VEL
LIN {X 0,Y 573.715,Z 295.239,A -85,B 0,C 180,E1 -2012.221,E2 -2012.221} C_VEL
LIN {X 0,Y 573.597,Z 305.781,A -85,B 0,C 180,E1 -2012.675,E2 -2012.675} C_VEL
LIN {X 0,Y 573.436,Z 316.517,A -85,B 0,C 180,E1 -2013.261,E2 -2013.261} C_VEL
LIN {X 0,Y 573.341,Z 328.757,A -85,B 0,C 180,E1 -2014.114,E2 -2014.114} C_VEL
LIN {X 0,Y 573.263,Z 338.283,A -85,B 0,C 180,E1 -2014.954,E2 -2014.954} C_VEL
LIN {X 0,Y 573.205,Z 346.217,A -85,B 0,C 180,E1 -2015.796,E2 -2015.796} C_VEL
LIN {X 0,Y 573.103,Z 353.42,A -85,B 0,C 180,E1 -2016.714,E2 -2016.714} C_VEL
LIN {X 0,Y 573.025,Z 359.446,A -85,B 0,C 180,E1 -2017.641,E2 -2017.641} C_VEL
LIN {X 0,Y 573.059,Z 365.125,A -85,B 0,C 180,E1 -2018.716,E2 -2018.716} C_VEL
LIN {X 0,Y 573.001,Z 370.504,A -85,B 0,C 180,E1 -2020.06,E2 -2020.06} C_VEL
LIN {X 0,Y 572.962,Z 373.274,A -85,B 0,C 180,E1 -2021.013,E2 -2021.013} C_VEL
LIN {X 0,Y 572.98,Z 375.893,A -85,B 0,C 180,E1 -2022.424,E2 -2022.424} C_VEL
LIN {X 0,Y 572.921,Z 376.885,A -85,B 0,C 180,E1 -2023.636,E2 -2023.636} C_VEL
LIN {X 0,Y 572.965,Z 376.802,A -85,B 0,C 180,E1 -2024.65,E2 -2024.65} C_VEL
LIN {X 0,Y 572.959,Z 375.925,A -85,B 0,C 180,E1 -2025.641,E2 -2025.641} C_VEL
LIN {X 0,Y 572.932,Z 374.286,A -85,B 0,C 180,E1 -2026.613,E2 -2026.613} C_VEL
LIN {X 0,Y 573.001,Z 371.863,A -85,B 0,C 180,E1 -2027.579,E2 -2027.579} C_VEL
LIN {X 0,Y 573.007,Z 368.696,A -85,B 0,C 180,E1 -2028.524,E2 -2028.524} C_VEL
LIN {X 0,Y 573.036,Z 364.512,A -85,B 0,C 180,E1 -2029.499,E2 -2029.499} C_VEL
LIN {X 0,Y 573.087,Z 358.611,A -85,B 0,C 180,E1 -2030.587,E2 -2030.587} C_VEL
LIN {X 0,Y 573.106,Z 352.381,A -85,B 0,C 180,E1 -2031.52,E2 -2031.52} C_VEL
LIN {X 0,Y 573.193,Z 344.111,A -85,B 0,C 180,E1 -2032.54,E2 -2032.54} C_VEL
LIN {X 0,Y 573.327,Z 334.165,A -85,B 0,C 180,E1 -2033.522,E2 -2033.522} C_VEL
LIN {X 0,Y 573.403,Z 324.44,A -85,B 0,C 180,E1 -2034.297,E2 -2034.297} C_VEL
LIN {X 0,Y 573.498,Z 314.677,A -85,B 0,C 180,E1 -2034.936,E2 -2034.936} C_VEL
LIN {X 0,Y 573.598,Z 305.483,A -85,B 0,C 180,E1 -2035.43,E2 -2035.43} C_VEL
LIN {X 0,Y 573.706,Z 294.639,A -85,B 0,C 180,E1 -2035.892,E2 -2035.892} C_VEL
LIN {X 0,Y 573.8,Z 282.498,A -85,B 0,C 180,E1 -2036.277,E2 -2036.277} C_VEL
LIN {X 0,Y 573.877,Z 269.68,A -85,B 0,C 180,E1 -2036.538,E2 -2036.538} C_VEL
LIN {X 0,Y 573.933,Z 170.062,A -85,B 0,C 180,E1 -2037.798,E2 -2037.798} C_VEL
LIN {X 0,Y 573.274,Z 166.126,A -85,B 0,C 180,E1 -2037.875,E2 -2037.875} C_VEL
LIN {X 0,Y 573.432,Z 148.993,A -85,B 0,C 180,E1 -2040.845,E2 -2040.845} C_VEL
LIN {X 0,Y 573.548,Z 134.251,A -85,B 0,C 180,E1 -2043.445,E2 -2043.445} C_VEL
LIN {X 0,Y 573.222,Z 132.083,A -85,B 0,C 180,E1 -2043.858,E2 -2043.858} C_VEL
LIN {X 0,Y 573.186,Z 132.085,A -85,B 0,C 180,E1 -2046.133,E2 -2046.133} C_VEL
LIN {X 0,Y 573.22,Z 132.079,A -85,B 0,C 180,E1 -2049.173,E2 -2049.173} C_VEL
LIN {X 0,Y 573.186,Z 132.081,A -85,B 0,C 180,E1 -2051.41,E2 -2051.41} C_VEL
LIN {X 0,Y 573.198,Z 132.088,A -85,B 0,C 180,E1 -2054.351,E2 -2054.351} C_VEL
LIN {X 0,Y 573.189,Z 132.088,A -85,B 0,C 180,E1 -2056.529,E2 -2056.529} C_VEL
LIN {X 0,Y 573.235,Z 132.075,A -85,B 0,C 180,E1 -2059.403,E2 -2059.403} C_VEL
LIN {X 0,Y 573.215,Z 132.087,A -85,B 0,C 180,E1 -2062.249,E2 -2062.249} C_VEL
LIN {X 0,Y 573.269,Z 132.071,A -85,B 0,C 180,E1 -2065.077,E2 -2065.077} C_VEL
LIN {X 0,Y 573.305,Z 132.072,A -85,B 0,C 180,E1 -2067.893,E2 -2067.893} C_VEL
LIN {X 0,Y 573.313,Z 132.073,A -85,B 0,C 180,E1 -2070,E2 -2070} C_VEL
LIN {X 0,Y 573.266,Z 132.071,A -85,B 0,C 180,E1 -2072.811,E2 -2072.811} C_VEL
LIN {X 0,Y 573.263,Z 132.076,A -85,B 0,C 180,E1 -2075.628,E2 -2075.628} C_VEL
LIN {X 0,Y 573.23,Z 132.077,A -85,B 0,C 180,E1 -2078.46,E2 -2078.46} C_VEL
LIN {X 0,Y 573.232,Z 132.077,A -85,B 0,C 180,E1 -2081.313,E2 -2081.313} C_VEL
LIN {X 0,Y 573.233,Z 132.076,A -85,B 0,C 180,E1 -2084.406,E2 -2084.406} C_VEL
LIN {X 0,Y 573.188,Z 132.082,A -85,B 0,C 180,E1 -2087.114,E2 -2087.114} C_VEL
LIN {X 0,Y 573.199,Z 132.082,A -85,B 0,C 180,E1 -2090.078,E2 -2090.078} C_VEL
LIN {X 0,Y 573.189,Z 132.081,A -85,B 0,C 180,E1 -2092.339,E2 -2092.339} C_VEL
LIN {X 0,Y 573.222,Z 132.085,A -85,B 0,C 180,E1 -2095.411,E2 -2095.411} C_VEL
LIN {X 0,Y 573.189,Z 132.082,A -85,B 0,C 180,E1 -2098.018,E2 -2098.018} C_VEL
LIN {X 0,Y 573.201,Z 132.081,A -85,B 0,C 180,E1 -2100.878,E2 -2100.878} C_VEL
LIN {X 0,Y 573.236,Z 132.081,A -85,B 0,C 180,E1 -2103.521,E2 -2103.521} C_VEL
LIN {X 0,Y 573.179,Z 132.082,A -85,B 0,C 180,E1 -2106.054,E2 -2106.054} C_VEL
LIN {X 0,Y 573.222,Z 132.079,A -85,B 0,C 180,E1 -2108.703,E2 -2108.703} C_VEL
LIN {X 0,Y 573.189,Z 132.084,A -85,B 0,C 180,E1 -2111.589,E2 -2111.589} C_VEL
LIN {X 0,Y 573.201,Z 132.083,A -85,B 0,C 180,E1 -2114.673,E2 -2114.673} C_VEL
LIN {X 0,Y 573.201,Z 132.081,A -85,B 0,C 180,E1 -2117.597,E2 -2117.597} C_VEL
LIN {X 0,Y 573.22,Z 132.079,A -85,B 0,C 180,E1 -2120.391,E2 -2120.391} C_VEL
LIN {X 0,Y 573.221,Z 132.083,A -85,B 0,C 180,E1 -2123.076,E2 -2123.076} C_VEL
LIN {X 0,Y 573.235,Z 132.075,A -85,B 0,C 180,E1 -2125.67,E2 -2125.67} C_VEL
LIN {X 0,Y 573.212,Z 132.079,A -85,B 0,C 180,E1 -2128.183,E2 -2128.183} C_VEL
LIN {X 0,Y 573.207,Z 132.087,A -85,B 0,C 180,E1 -2130.631,E2 -2130.631} C_VEL
LIN {X 0,Y 573.197,Z 132.08,A -85,B 0,C 180,E1 -2133.514,E2 -2133.514} C_VEL
LIN {X 0,Y 573.184,Z 132.084,A -85,B 0,C 180,E1 -2136.133,E2 -2136.133} C_VEL
LIN {X 0,Y 573.218,Z 132.078,A -85,B 0,C 180,E1 -2139.173,E2 -2139.173} C_VEL
LIN {X 0,Y 573.183,Z 132.081,A -85,B 0,C 180,E1 -2141.41,E2 -2141.41} C_VEL
LIN {X 0,Y 573.195,Z 132.089,A -85,B 0,C 180,E1 -2144.351,E2 -2144.351} C_VEL
LIN {X 0,Y 573.186,Z 132.088,A -85,B 0,C 180,E1 -2146.529,E2 -2146.529} C_VEL
LIN {X 0,Y 573.232,Z 132.075,A -85,B 0,C 180,E1 -2149.403,E2 -2149.403} C_VEL
LIN {X 0,Y 573.211,Z 132.088,A -85,B 0,C 180,E1 -2152.249,E2 -2152.249} C_VEL
LIN {X 0,Y 573.266,Z 132.071,A -85,B 0,C 180,E1 -2155.077,E2 -2155.077} C_VEL
LIN {X 0,Y 573.303,Z 132.073,A -85,B 0,C 180,E1 -2157.893,E2 -2157.893} C_VEL
LIN {X 0,Y 573.31,Z 132.074,A -85,B 0,C 180,E1 -2160,E2 -2160} C_VEL
LIN {X 0,Y 573.263,Z 132.072,A -85,B 0,C 180,E1 -2162.811,E2 -2162.811} C_VEL
LIN {X 0,Y 573.261,Z 132.076,A -85,B 0,C 180,E1 -2165.629,E2 -2165.629} C_VEL
LIN {X 0,Y 573.227,Z 132.077,A -85,B 0,C 180,E1 -2168.461,E2 -2168.461} C_VEL
LIN {X 0,Y 573.229,Z 132.078,A -85,B 0,C 180,E1 -2171.313,E2 -2171.313} C_VEL
LIN {X 0,Y 573.23,Z 132.076,A -85,B 0,C 180,E1 -2174.406,E2 -2174.406} C_VEL
LIN {X 0,Y 573.185,Z 132.083,A -85,B 0,C 180,E1 -2177.114,E2 -2177.114} C_VEL
LIN {X 0,Y 573.197,Z 132.082,A -85,B 0,C 180,E1 -2180.079,E2 -2180.079} C_VEL
LIN {X 0,Y 573.188,Z 132.081,A -85,B 0,C 180,E1 -2182.34,E2 -2182.34} C_VEL
LIN {X 0,Y 573.22,Z 132.085,A -85,B 0,C 180,E1 -2185.412,E2 -2185.412} C_VEL
LIN {X 0,Y 573.188,Z 132.082,A -85,B 0,C 180,E1 -2188.018,E2 -2188.018} C_VEL
LIN {X 0,Y 573.198,Z 132.082,A -85,B 0,C 180,E1 -2190.878,E2 -2190.878} C_VEL
LIN {X 0,Y 573.238,Z 132.081,A -85,B 0,C 180,E1 -2193.521,E2 -2193.521} C_VEL
LIN {X 0,Y 573.177,Z 132.082,A -85,B 0,C 180,E1 -2196.055,E2 -2196.055} C_VEL
LIN {X 0,Y 573.223,Z 132.079,A -85,B 0,C 180,E1 -2198.703,E2 -2198.703} C_VEL
LIN {X 0,Y 573.191,Z 132.083,A -85,B 0,C 180,E1 -2201.589,E2 -2201.589} C_VEL
LIN {X 0,Y 573.205,Z 132.082,A -85,B 0,C 180,E1 -2204.674,E2 -2204.674} C_VEL
LIN {X 0,Y 573.201,Z 132.08,A -85,B 0,C 180,E1 -2207.597,E2 -2207.597} C_VEL
LIN {X 0,Y 573.228,Z 132.08,A -85,B 0,C 180,E1 -2210.571,E2 -2210.571} C_VEL
LIN {X 0,Y 573.224,Z 132.083,A -85,B 0,C 180,E1 -2213.076,E2 -2213.076} C_VEL
LIN {X 0,Y 573.238,Z 132.074,A -85,B 0,C 180,E1 -2215.67,E2 -2215.67} C_VEL
LIN {X 0,Y 573.205,Z 132.08,A -85,B 0,C 180,E1 -2218.183,E2 -2218.183} C_VEL
LIN {X 0,Y 573.212,Z 132.087,A -85,B 0,C 180,E1 -2220.632,E2 -2220.632} C_VEL
LIN {X 0,Y 573.193,Z 132.08,A -85,B 0,C 180,E1 -2223.517,E2 -2223.517} C_VEL
LIN {X 0,Y 573.188,Z 132.085,A -85,B 0,C 180,E1 -2226.133,E2 -2226.133} C_VEL
LIN {X 0,Y 573.22,Z 132.185,A -85,B 0,C 180,E1 -2226.984,E2 -2226.984} C_VEL
LIN {X 0,Y 573.885,Z 136.732,A -85,B 0,C 180,E1 -2227.689,E2 -2227.689} C_VEL
LIN {X 0,Y 573.754,Z 154.542,A -85,B 0,C 180,E1 -2230.315,E2 -2230.315} C_VEL
LIN {X 0,Y 573.542,Z 173.143,A -85,B 0,C 180,E1 -2233.023,E2 -2233.023} C_VEL
LIN {X 0,Y 573.405,Z 193.691,A -85,B 0,C 180,E1 -2235.991,E2 -2235.991} C_VEL
LIN {X 0,Y 573.402,Z 195.149,A -85,B 0,C 180,E1 -2236.172,E2 -2236.172} C_VEL
LIN {X 0,Y 574.052,Z 200.515,A -85,B 0,C 180,E1 -2236.256,E2 -2236.256} C_VEL
LIN {X 0,Y 573.887,Z 302.95,A -85,B 0,C 180,E1 -2237.558,E2 -2237.558} C_VEL
LIN {X 0,Y 573.778,Z 316.22,A -85,B 0,C 180,E1 -2237.869,E2 -2237.869} C_VEL
LIN {X 0,Y 573.699,Z 328.378,A -85,B 0,C 180,E1 -2238.294,E2 -2238.294} C_VEL
LIN {X 0,Y 573.589,Z 339.602,A -85,B 0,C 180,E1 -2238.818,E2 -2238.818} C_VEL
LIN {X 0,Y 573.456,Z 350.907,A -85,B 0,C 180,E1 -2239.496,E2 -2239.496} C_VEL
LIN {X 0,Y 573.35,Z 361.54,A -85,B 0,C 180,E1 -2240.297,E2 -2240.297} C_VEL
LIN {X 0,Y 573.241,Z 371.113,A -85,B 0,C 180,E1 -2241.185,E2 -2241.185} C_VEL
LIN {X 0,Y 573.161,Z 378.961,A -85,B 0,C 180,E1 -2242.071,E2 -2242.071} C_VEL
LIN {X 0,Y 573.073,Z 386.955,A -85,B 0,C 180,E1 -2243.185,E2 -2243.185} C_VEL
LIN {X 0,Y 573.07,Z 393.68,A -85,B 0,C 180,E1 -2244.37,E2 -2244.37} C_VEL
LIN {X 0,Y 573.028,Z 398.372,A -85,B 0,C 180,E1 -2245.427,E2 -2245.427} C_VEL
LIN {X 0,Y 573.022,Z 401.957,A -85,B 0,C 180,E1 -2246.484,E2 -2246.484} C_VEL
LIN {X 0,Y 572.959,Z 403.808,A -85,B 0,C 180,E1 -2247.188,E2 -2247.188} C_VEL
LIN {X 0,Y 572.946,Z 406.185,A -85,B 0,C 180,E1 -2248.594,E2 -2248.594} C_VEL
LIN {X 0,Y 572.938,Z 407,A -85,B 0,C 180,E1 -2250,E2 -2250} C_VEL
LIN {X 0,Y 572.946,Z 406.186,A -85,B 0,C 180,E1 -2251.406,E2 -2251.406} C_VEL
LIN {X 0,Y 572.94,Z 405.199,A -85,B 0,C 180,E1 -2252.109,E2 -2252.109} C_VEL
LIN {X 0,Y 572.959,Z 403.81,A -85,B 0,C 180,E1 -2252.812,E2 -2252.812} C_VEL
LIN {X 0,Y 573.015,Z 400.896,A -85,B 0,C 180,E1 -2253.868,E2 -2253.868} C_VEL
LIN {X 0,Y 572.963,Z 396.949,A -85,B 0,C 180,E1 -2254.925,E2 -2254.925} C_VEL
LIN {X 0,Y 573.065,Z 390.878,A -85,B 0,C 180,E1 -2256.16,E2 -2256.16} C_VEL
LIN {X 0,Y 573.119,Z 384.238,A -85,B 0,C 180,E1 -2257.221,E2 -2257.221} C_VEL
LIN {X 0,Y 573.201,Z 375.993,A -85,B 0,C 180,E1 -2258.283,E2 -2258.283} C_VEL
LIN {X 0,Y 573.287,Z 367.542,A -85,B 0,C 180,E1 -2259.17,E2 -2259.17} C_VEL
LIN {X 0,Y 573.427,Z 357.099,A -85,B 0,C 180,E1 -2260.058,E2 -2260.058} C_VEL
LIN {X 0,Y 573.543,Z 345.436,A -85,B 0,C 180,E1 -2260.853,E2 -2260.853} C_VEL
LIN {X 0,Y 573.651,Z 334.313,A -85,B 0,C 180,E1 -2261.446,E2 -2261.446} C_VEL
LIN {X 0,Y 573.758,Z 321.178,A -85,B 0,C 180,E1 -2261.974,E2 -2261.974} C_VEL
LIN {X 0,Y 573.855,Z 308.529,A -85,B 0,C 180,E1 -2262.331,E2 -2262.331} C_VEL
